   t1[3799] := 0.1576416;
   t1[3800] := 0.1064425;
   t1[3801] := 0.0526067;
   t1[3802] := -0.0066586;
   t1[3803] := -0.0740744;
   t1[3804] := -0.1487714;
   t1[3805] := -0.2246916;
   t1[3806] := -0.2953722;
   t1[3807] := -0.3543501;
   t1[3808] := -0.3951623;
   t1[3809] := -0.4124203;
   t1[3810] := 0.2382786;
   t1[3811] := 0.2234323;
   t1[3812] := 0.2057212;
   t1[3813] := 0.1861852;
   t1[3814] := 0.1646943;
   t1[3815] := 0.1407051;
   t1[3816] := 0.1136735;
   t1[3817] := 0.0830556;
   t1[3818] := 0.0483291;
   t1[3819] := 0.0100414;
   t1[3820] := -0.0297129;
   t1[3821] := -0.0687187;
   t1[3822] := -0.1047607;
   t1[3823] := -0.1356239;
   t1[3824] := -0.1593218;
   t1[3825] := 0.0314255;
   t1[3826] := 0.0159087;
   t1[3827] := 0.0083954;
   t1[3828] := 0.0117159;
   t1[3829] := 0.0246836;
   t1[3830] := 0.0446926;
   t1[3831] := 0.0691354;
   t1[3832] := 0.0954045;
   t1[3833] := 0.1209108;
   t1[3834] := 0.1439967;
   t1[3835] := 0.1643503;
   t1[3836] := 0.1817647;
   t1[3837] := 0.1960331;
   t1[3838] := 0.2069486;
   t1[3839] := 0.2142785;
   t1[3840] := 0.0667891;
   t1[3841] := 0.0459893;
   t1[3842] := 0.0290749;
   t1[3843] := 0.0181673;
   t1[3844] := 0.0125522;
   t1[3845] := 0.0105136;
   t1[3846] := 0.010334;
   t1[3847] := 0.0102961;
   t1[3848] := 0.0087127;
   t1[3849] := 0.0054041;
   t1[3850] := 0.0023689;
   t1[3851] := 0.0017762;
   t1[3852] := 0.0057949;
   t1[3853] := 0.0165937;
   t1[3854] := 0.0358182;
   t1[3855] := -0.1236024;
   t1[3856] := -0.1436511;
   t1[3857] := -0.1554508;
   t1[3858] := -0.1564814;
   t1[3859] := -0.1472676;
   t1[3860] := -0.1294098;
   t1[3861] := -0.1045099;
   t1[3862] := -0.0741695;
   t1[3863] := -0.0400035;
   t1[3864] := -0.0042752;
   t1[3865] := 0.029814;
   t1[3866] := 0.05899;
   t1[3867] := 0.0799781;
   t1[3868] := 0.0895042;
   t1[3869] := 0.0849915;
   t1[3870] := 0.1448045;
   t1[3871] := 0.1536896;
   t1[3872] := 0.1602021;
   t1[3873] := 0.1635016;
   t1[3874] := 0.1634868;
   t1[3875] := 0.1603173;
   t1[3876] := 0.1541528;
   t1[3877] := 0.1451532;
   t1[3878] := 0.1334766;
   t1[3879] := 0.1191958;
   t1[3880] := 0.1022594;
   t1[3881] := 0.0826069;
   t1[3882] := 0.0601774;
   t1[3883] := 0.0349101;
   t1[3884] := 0.0069634;
   t1[3885] := 0.0060057;
   t1[3886] := -0.002674;
   t1[3887] := -0.0069002;
   t1[3888] := -0.0053898;
   t1[3889] := 0.001487;
   t1[3890] := 0.0127761;
   t1[3891] := 0.0275223;
   t1[3892] := 0.0447709;
   t1[3893] := 0.063564;
   t1[3894] := 0.0828049;
   t1[3895] := 0.1011957;
   t1[3896] := 0.1174229;
   t1[3897] := 0.130173;
   t1[3898] := 0.1381326;
   t1[3899] := 0.1401622;
   t1[3900] := 0.1874084;
   t1[3901] := 0.1562083;
   t1[3902] := 0.1240833;
   t1[3903] := 0.0933504;
   t1[3904] := 0.0642;
   t1[3905] := 0.0360715;
   t1[3906] := 0.0084033;
   t1[3907] := -0.0193662;
   t1[3908] := -0.0477891;
   t1[3909] := -0.0769431;
   t1[3910] := -0.1062206;
   t1[3911] := -0.1349603;
   t1[3912] := -0.162501;
   t1[3913] := -0.1881814;
   t1[3914] := -0.2112326;
   t1[3915] := -0.0535974;
   t1[3916] := -0.0502168;
   t1[3917] := -0.0400993;
   t1[3918] := -0.0239367;
   t1[3919] := -0.0041446;
   t1[3920] := 0.0162519;
   t1[3921] := 0.0342271;
   t1[3922] := 0.0467551;
   t1[3923] := 0.0508583;
   t1[3924] := 0.0459583;
   t1[3925] := 0.0349444;
   t1[3926] := 0.0209767;
   t1[3927] := 0.0072152;
   t1[3928] := -0.0031799;
   t1[3929] := -0.0075761;
   t1[3930] := 0.1498998;
   t1[3931] := 0.130271;
   t1[3932] := 0.107127;
   t1[3933] := 0.0806729;
   t1[3934] := 0.052375;
   t1[3935] := 0.0241449;
   t1[3936] := -0.0021051;
   t1[3937] := -0.0244629;
   t1[3938] := -0.0410386;
   t1[3939] := -0.0510728;
   t1[3940] := -0.0554392;
   t1[3941] := -0.055139;
   t1[3942] := -0.0511733;
   t1[3943] := -0.0445433;
   t1[3944] := -0.0362266;
   t1[3945] := -0.2330382;
   t1[3946] := -0.1871568;
   t1[3947] := -0.1450667;
   t1[3948] := -0.1113965;
   t1[3949] := -0.0854538;
   t1[3950] := -0.0646658;
   t1[3951] := -0.0464576;
   t1[3952] := -0.0282541;
   t1[3953] := -0.0075134;
   t1[3954] := 0.0166584;
   t1[3955] := 0.0427734;
   t1[3956] := 0.0691579;
   t1[3957] := 0.0941378;
   t1[3958] := 0.1160396;
   t1[3959] := 0.1332923;
   t1[3960] := -0.0491654;
   t1[3961] := -0.036231;
   t1[3962] := -0.0223325;
   t1[3963] := -0.0065351;
   t1[3964] := 0.0112607;
   t1[3965] := 0.0308597;
   t1[3966] := 0.0520663;
   t1[3967] := 0.0746847;
   t1[3968] := 0.0985081;
   t1[3969] := 0.1227671;
   t1[3970] := 0.1458796;
   t1[3971] := 0.1662;
   t1[3972] := 0.1820826;
   t1[3973] := 0.1918821;
   t1[3974] := 0.1942146;
   t1[3975] := -0.0419469;
   t1[3976] := -0.024382;
   t1[3977] := -0.0039275;
   t1[3978] := 0.0193405;
   t1[3979] := 0.043617;
   t1[3980] := 0.0664858;
   t1[3981] := 0.0855298;
   t1[3982] := 0.0983321;
   t1[3983] := 0.1025108;
   t1[3984] := 0.0974387;
   t1[3985] := 0.0850243;
   t1[3986] := 0.0673741;
   t1[3987] := 0.0465946;
   t1[3988] := 0.0247923;
   t1[3989] := 0.0039388;
   t1[3990] := 0.081306;
   t1[3991] := 0.0967213;
   t1[3992] := 0.1059721;
   t1[3993] := 0.105438;
   t1[3994] := 0.0966705;
   t1[3995] := 0.0830483;
   t1[3996] := 0.067952;
   t1[3997] := 0.0547624;
   t1[3998] := 0.0468165;
   t1[3999] := 0.0452519;
   t1[4000] := 0.0480284;
   t1[4001] := 0.0528576;
   t1[4002] := 0.0574511;
   t1[4003] := 0.0595205;
   t1[4004] := 0.0571091;
   t1[4005] := -0.3532258;
   t1[4006] := -0.347388;
   t1[4007] := -0.3259861;
   t1[4008] := -0.2866082;
   t1[4009] := -0.2320336;
   t1[4010] := -0.1668758;
   t1[4011] := -0.0957504;
   t1[4012] := -0.023273;
   t1[4013] := 0.0459573;
   t1[4014] := 0.1081692;
   t1[4015] := 0.1607873;
   t1[4016] := 0.2013298;
   t1[4017] := 0.2273147;
   t1[4018] := 0.2362603;
   t1[4019] := 0.2265386;
   t1[4020] := -0.1837068;
   t1[4021] := -0.1607816;
   t1[4022] := -0.1328929;
   t1[4023] := -0.1009052;
   t1[4024] := -0.066294;
   t1[4025] := -0.0307508;
   t1[4026] := 0.004033;
   t1[4027] := 0.0363657;
   t1[4028] := 0.064572;
   t1[4029] := 0.0877905;
   t1[4030] := 0.1063364;
   t1[4031] := 0.1206166;
   t1[4032] := 0.1310381;
   t1[4033] := 0.1380079;
   t1[4034] := 0.1419902;
   t1[4035] := 0.1791124;
   t1[4036] := 0.1800564;
   t1[4037] := 0.179791;
   t1[4038] := 0.1790846;
   t1[4039] := 0.1772211;
   t1[4040] := 0.1729594;
   t1[4041] := 0.1650582;
   t1[4042] := 0.1522758;
   t1[4043] := 0.133402;
   t1[4044] := 0.1087973;
   t1[4045] := 0.0810914;
   t1[4046] := 0.0530913;
   t1[4047] := 0.027604;
   t1[4048] := 0.0074365;
   t1[4049] := -0.0050674;
   t1[4050] := 0.18974;
   t1[4051] := 0.1681934;
   t1[4052] := 0.1429099;
   t1[4053] := 0.115058;
   t1[4054] := 0.0845972;
   t1[4055] := 0.0510596;
   t1[4056] := 0.0139768;
   t1[4057] := -0.0271196;
   t1[4058] := -0.0726646;
   t1[4059] := -0.1214214;
   t1[4060] := -0.1697376;
   t1[4061] := -0.2137718;
   t1[4062] := -0.249683;
   t1[4063] := -0.27363;
   t1[4064] := -0.282454;
   t1[4065] := -0.0203979;
   t1[4066] := -0.0223091;
   t1[4067] := -0.0231968;
   t1[4068] := -0.0224718;
   t1[4069] := -0.0193559;
   t1[4070] := -0.0130042;
   t1[4071] := -0.0025716;
   t1[4072] := 0.012787;
   t1[4073] := 0.0338832;
   t1[4074] := 0.05985;
   t1[4075] := 0.0873946;
   t1[4076] := 0.113035;
   t1[4077] := 0.1332889;
   t1[4078] := 0.1446745;
   t1[4079] := 0.1443445;
   t1[4080] := 0.058554;
   t1[4081] := 0.0751369;
   t1[4082] := 0.0861599;
   t1[4083] := 0.0897582;
   t1[4084] := 0.0872719;
   t1[4085] := 0.0811738;
   t1[4086] := 0.0739379;
   t1[4087] := 0.0680383;
   t1[4088] := 0.0659192;
   t1[4089] := 0.068534;
   t1[4090] := 0.0746809;
   t1[4091] := 0.0829904;
   t1[4092] := 0.0920926;
   t1[4093] := 0.1006178;
   t1[4094] := 0.1072876;
   t1[4095] := -0.1914829;
   t1[4096] := -0.137766;
   t1[4097] := -0.0834525;
   t1[4098] := -0.0324906;
   t1[4099] := 0.0136321;
   t1[4100] := 0.0542972;
   t1[4101] := 0.0888875;
   t1[4102] := 0.1167857;
   t1[4103] := 0.1373913;
   t1[4104] := 0.1509367;
   t1[4105] := 0.1588583;
   t1[4106] := 0.1626864;
   t1[4107] := 0.1639515;
   t1[4108] := 0.164184;
   t1[4109] := 0.1646439;
   t1[4110] := -0.0583478;
   t1[4111] := -0.0186663;
   t1[4112] := 0.0169952;
   t1[4113] := 0.04533;
   t1[4114] := 0.0669303;
   t1[4115] := 0.0837658;
   t1[4116] := 0.0978078;
   t1[4117] := 0.1110275;
   t1[4118] := 0.1253682;
   t1[4119] := 0.1413658;
   t1[4120] := 0.1575224;
   t1[4121] := 0.1721816;
   t1[4122] := 0.1836867;
   t1[4123] := 0.1903812;
   t1[4124] := 0.190859;
   t1[4125] := -0.0328098;
   t1[4126] := -0.0068127;
   t1[4127] := 0.0114748;
   t1[4128] := 0.0191703;
   t1[4129] := 0.0181671;
   t1[4130] := 0.0120459;
   t1[4131] := 0.0043894;
   t1[4132] := -0.0012196;
   t1[4133] := -0.0012441;
   t1[4134] := 0.0055699;
   t1[4135] := 0.0171766;
   t1[4136] := 0.0312727;
   t1[4137] := 0.0455549;
   t1[4138] := 0.05772;
   t1[4139] := 0.0657464;
   t1[4140] := 0.0864437;
   t1[4141] := 0.0887006;
   t1[4142] := 0.0839517;
   t1[4143] := 0.0726865;
   t1[4144] := 0.0565655;
   t1[4145] := 0.0376631;
   t1[4146] := 0.018054;
   t1[4147] := -0.0001868;
   t1[4148] := -0.0150103;
   t1[4149] := -0.0256528;
   t1[4150] := -0.0332085;
   t1[4151] := -0.0389166;
   t1[4152] := -0.0440164;
   t1[4153] := -0.049747;
   t1[4154] := -0.0571015;
   t1[4155] := -0.0806194;
   t1[4156] := -0.0510695;
   t1[4157] := -0.0227195;
   t1[4158] := 0.0029388;
   t1[4159] := 0.0255656;
   t1[4160] := 0.0452287;
   t1[4161] := 0.0619963;
   t1[4162] := 0.0759363;
   t1[4163] := 0.0871133;
   t1[4164] := 0.0954085;
   t1[4165] := 0.1004382;
   t1[4166] := 0.1017982;
   t1[4167] := 0.0990841;
   t1[4168] := 0.0918918;
   t1[4169] := 0.080022;
   t1[4170] := 0.0758055;
   t1[4171] := 0.0483579;
   t1[4172] := 0.019726;
   t1[4173] := -0.0085936;
   t1[4174] := -0.0351953;
   t1[4175] := -0.0587056;
   t1[4176] := -0.0777511;
   t1[4177] := -0.0909582;
   t1[4178] := -0.0969803;
   t1[4179] := -0.0958076;
   t1[4180] := -0.0893632;
   t1[4181] := -0.0797205;
   t1[4182] := -0.0689533;
   t1[4183] := -0.0591352;
   t1[4184] := -0.0520488;
   t1[4185] := 0.0500193;
   t1[4186] := 0.0250257;
   t1[4187] := 0.0067496;
   t1[4188] := -0.0013496;
   t1[4189] := -0.0002283;
   t1[4190] := 0.0075968;
   t1[4191] := 0.0196071;
   t1[4192] := 0.0332839;
   t1[4193] := 0.0461257;
   t1[4194] := 0.0564741;
   t1[4195] := 0.06389;
   t1[4196] := 0.0680293;
   t1[4197] := 0.0685479;
   t1[4198] := 0.0651018;
   t1[4199] := 0.0575236;
   t1[4200] := -0.1111487;
   t1[4201] := -0.1043046;
   t1[4202] := -0.0834341;
   t1[4203] := -0.0456349;
   t1[4204] := 0.0052346;
   t1[4205] := 0.0629264;
   t1[4206] := 0.1211901;
   t1[4207] := 0.1737752;
   t1[4208] := 0.2144941;
   t1[4209] := 0.2403017;
   t1[4210] := 0.2526951;
   t1[4211] := 0.2535257;
   t1[4212] := 0.2446451;
   t1[4213] := 0.2279048;
   t1[4214] := 0.2051906;
   t1[4215] := -0.1796006;
   t1[4216] := -0.1449579;
   t1[4217] := -0.1035627;
   t1[4218] := -0.0561289;
   t1[4219] := -0.0046341;
   t1[4220] := 0.0484977;
   t1[4221] := 0.1008417;
   t1[4222] := 0.1499734;
   t1[4223] := 0.1934813;
   t1[4224] := 0.229624;
   t1[4225] := 0.2576274;
   t1[4226] := 0.2767932;
   t1[4227] := 0.2864232;
   t1[4228] := 0.285819;
   t1[4229] := 0.2745421;
   t1[4230] := -0.1943461;
   t1[4231] := -0.1704851;
   t1[4232] := -0.1405829;
   t1[4233] := -0.1052732;
   t1[4234] := -0.0649546;
   t1[4235] := -0.0199427;
   t1[4236] := 0.0294473;
   t1[4237] := 0.0828997;
   t1[4238] := 0.1400708;
   t1[4239] := 0.1992041;
   t1[4240] := 0.2565007;
   t1[4241] := 0.3080023;
   t1[4242] := 0.3497505;
   t1[4243] := 0.3777874;
   t1[4244] := 0.3887276;
   t1[4245] := 0.1895632;
   t1[4246] := 0.1862952;
   t1[4247] := 0.1769894;
   t1[4248] := 0.1617853;
   t1[4249] := 0.1431127;
   t1[4250] := 0.1242102;
   t1[4251] := 0.1083174;
   t1[4252] := 0.0986739;
   t1[4253] := 0.0984564;
   t1[4254] := 0.1076931;
   t1[4255] := 0.1218616;
   t1[4256] := 0.1360845;
   t1[4257] := 0.145484;
   t1[4258] := 0.1451829;
   t1[4259] := 0.1312412;
   t1[4260] := -0.0941189;
   t1[4261] := -0.0750441;
   t1[4262] := -0.0494044;
   t1[4263] := -0.0175561;
   t1[4264] := 0.018117;
   t1[4265] := 0.0545142;
   t1[4266] := 0.0885344;
   t1[4267] := 0.117076;
   t1[4268] := 0.1370689;
   t1[4269] := 0.1470022;
   t1[4270] := 0.1476181;
   t1[4271] := 0.1398349;
   t1[4272] := 0.1245708;
   t1[4273] := 0.1027442;
   t1[4274] := 0.0753431;
   t1[4275] := 0.0685778;
   t1[4276] := 0.051928;
   t1[4277] := 0.0314925;
   t1[4278] := 0.007498;
   t1[4279] := -0.0187296;
   t1[4280] := -0.0454757;
   t1[4281] := -0.0710255;
   t1[4282] := -0.0936643;
   t1[4283] := -0.1116789;
   t1[4284] := -0.1234511;
   t1[4285] := -0.1274992;
   t1[4286] := -0.1223522;
   t1[4287] := -0.106539;
   t1[4288] := -0.0785887;
   t1[4289] := -0.0377033;
   t1[4290] := -0.1350671;
   t1[4291] := -0.1060196;
   t1[4292] := -0.0778034;
   t1[4293] := -0.0545455;
   t1[4294] := -0.0360641;
   t1[4295] := -0.020655;
   t1[4296] := -0.0066124;
   t1[4297] := 0.0077697;
   t1[4298] := 0.0241794;
   t1[4299] := 0.043411;
   t1[4300] := 0.0649677;
   t1[4301] := 0.0882515;
   t1[4302] := 0.1126646;
   t1[4303] := 0.1376094;
   t1[4304] := 0.1623792;
   t1[4305] := -0.0144924;
   t1[4306] := -0.0096911;
   t1[4307] := -0.00347;
   t1[4308] := 0.0033079;
   t1[4309] := 0.0099354;
   t1[4310] := 0.0157605;
   t1[4311] := 0.0201311;
   t1[4312] := 0.022395;
   t1[4313] := 0.0219254;
   t1[4314] := 0.0193535;
   t1[4315] := 0.0171285;
   t1[4316] := 0.0178418;
   t1[4317] := 0.0240846;
   t1[4318] := 0.0384482;
   t1[4319] := 0.0627826;
   t1[4320] := -0.1042536;
   t1[4321] := -0.0667104;
   t1[4322] := -0.0323665;
   t1[4323] := -0.0045362;
   t1[4324] := 0.017397;
   t1[4325] := 0.0354384;
   t1[4326] := 0.0515946;
   t1[4327] := 0.0678727;
   t1[4328] := 0.0862458;
   t1[4329] := 0.1070016;
   t1[4330] := 0.1279919;
   t1[4331] := 0.1468786;
   t1[4332] := 0.1613233;
   t1[4333] := 0.1689879;
   t1[4334] := 0.1679946;
   t1[4335] := 0.0434848;
   t1[4336] := 0.0531504;
   t1[4337] := 0.0601945;
   t1[4338] := 0.0632927;
   t1[4339] := 0.0616237;
   t1[4340] := 0.0545442;
   t1[4341] := 0.0414107;
   t1[4342] := 0.0215801;
   t1[4343] := -0.0055602;
   t1[4344] := -0.0390802;
   t1[4345] := -0.0758206;
   t1[4346] := -0.1124483;
   t1[4347] := -0.1456301;
   t1[4348] := -0.1720328;
   t1[4349] := -0.1887759;
   t1[4350] := -0.0447853;
   t1[4351] := -0.0387455;
   t1[4352] := -0.0276729;
   t1[4353] := -0.0104063;
   t1[4354] := 0.0118896;
   t1[4355] := 0.0372285;
   t1[4356] := 0.0636228;
   t1[4357] := 0.0890853;
   t1[4358] := 0.1116374;
   t1[4359] := 0.1297481;
   t1[4360] := 0.1425325;
   t1[4361] := 0.1491565;
   t1[4362] := 0.1487859;
   t1[4363] := 0.1405863;
   t1[4364] := 0.1241035;
   t1[4365] := 0.1752176;
   t1[4366] := 0.1764574;
   t1[4367] := 0.1733454;
   t1[4368] := 0.166352;
   t1[4369] := 0.1567683;
   t1[4370] := 0.1461753;
   t1[4371] := 0.1361545;
   t1[4372] := 0.1282874;
   t1[4373] := 0.1241305;
   t1[4374] := 0.1239933;
   t1[4375] := 0.1263832;
   t1[4376] := 0.1296669;
   t1[4377] := 0.1322112;
   t1[4378] := 0.1323828;
   t1[4379] := 0.1288362;
   t1[4380] := 0.1311117;
   t1[4381] := 0.1251942;
   t1[4382] := 0.1175675;
   t1[4383] := 0.1089724;
   t1[4384] := 0.100168;
   t1[4385] := 0.0919197;
   t1[4386] := 0.084993;
   t1[4387] := 0.0801534;
   t1[4388] := 0.0781383;
   t1[4389] := 0.0782922;
   t1[4390] := 0.0779461;
   t1[4391] := 0.0742737;
   t1[4392] := 0.0644488;
   t1[4393] := 0.0456451;
   t1[4394] := 0.015853;
   t1[4395] := 0.1653865;
   t1[4396] := 0.1615747;
   t1[4397] := 0.1489204;
   t1[4398] := 0.1252114;
   t1[4399] := 0.0928236;
   t1[4400] := 0.0557549;
   t1[4401] := 0.0180047;
   t1[4402] := -0.0164276;
   t1[4403] := -0.0435795;
   t1[4404] := -0.061344;
   t1[4405] := -0.0702954;
   t1[4406] := -0.0712172;
   t1[4407] := -0.0648929;
   t1[4408] := -0.0521063;
   t1[4409] := -0.033843;
   t1[4410] := -0.1095109;
   t1[4411] := -0.1050676;
   t1[4412] := -0.0937962;
   t1[4413] := -0.0753762;
   t1[4414] := -0.0512059;
   t1[4415] := -0.0232909;
   t1[4416] := 0.0063625;
   t1[4417] := 0.0357481;
   t1[4418] := 0.0628728;
   t1[4419] := 0.0864108;
   t1[4420] := 0.1059999;
   t1[4421] := 0.1213535;
   t1[4422] := 0.1321848;
   t1[4423] := 0.1382072;
   t1[4424] := 0.1392217;
   t1[4425] := 0.1267594;
   t1[4426] := 0.1530687;
   t1[4427] := 0.1682366;
   t1[4428] := 0.1672206;
   t1[4429] := 0.1514878;
   t1[4430] := 0.1248052;
   t1[4431] := 0.0909425;
   t1[4432] := 0.0536695;
   t1[4433] := 0.0167313;
   t1[4434] := -0.0173527;
   t1[4435] := -0.047835;
   t1[4436] := -0.0741062;
   t1[4437] := -0.0955572;
   t1[4438] := -0.1115787;
   t1[4439] := -0.121677;
   t1[4440] := 0.0897872;
   t1[4441] := 0.0856847;
   t1[4442] := 0.0806051;
   t1[4443] := 0.0744163;
   t1[4444] := 0.0680452;
   t1[4445] := 0.0627932;
   t1[4446] := 0.0599619;
   t1[4447] := 0.060853;
   t1[4448] := 0.0667383;
   t1[4449] := 0.0773905;
   t1[4450] := 0.0904158;
   t1[4451] := 0.1032513;
   t1[4452] := 0.113334;
   t1[4453] := 0.1181012;
   t1[4454] := 0.115397;
   t1[4455] := 0.1432041;
   t1[4456] := 0.1568891;
   t1[4457] := 0.1634402;
   t1[4458] := 0.1613314;
   t1[4459] := 0.1513807;
   t1[4460] := 0.1352343;
   t1[4461] := 0.1145394;
   t1[4462] := 0.0909433;
   t1[4463] := 0.0660909;
   t1[4464] := 0.0415152;
   t1[4465] := 0.0185874;
   t1[4466] := -0.0013338;
   t1[4467] := -0.0168899;
   t1[4468] := -0.0267222;
   t1[4469] := -0.0297787;
   t1[4470] := -0.3758105;
   t1[4471] := -0.322452;
   t1[4472] := -0.2597182;
   t1[4473] := -0.1912154;
   t1[4474] := -0.1200375;
   t1[4475] := -0.049098;
   t1[4476] := 0.0186902;
   t1[4477] := 0.080414;
   t1[4478] := 0.1331862;
   t1[4479] := 0.1754149;
   t1[4480] := 0.20738;
   t1[4481] := 0.2295079;
   t1[4482] := 0.2422246;
   t1[4483] := 0.2459562;
   t1[4484] := 0.2412414;
   t1[4485] := -0.083162;
   t1[4486] := -0.068404;
   t1[4487] := -0.051038;
   t1[4488] := -0.032456;
   t1[4489] := -0.0130457;
   t1[4490] := 0.00716;
   t1[4491] := 0.0281286;
   t1[4492] := 0.0498277;
   t1[4493] := 0.072215;
   t1[4494] := 0.094764;
   t1[4495] := 0.1162474;
   t1[4496] := 0.1353838;
   t1[4497] := 0.1508913;
   t1[4498] := 0.1614884;
   t1[4499] := 0.1660409;
   t1[4500] := 0.1987849;
   t1[4501] := 0.1696371;
   t1[4502] := 0.1381494;
   t1[4503] := 0.1057929;
   t1[4504] := 0.0741976;
   t1[4505] := 0.0450496;
   t1[4506] := 0.0200352;
   t1[4507] := 0.0008408;
   t1[4508] := -0.010889;
   t1[4509] := -0.0155813;
   t1[4510] := -0.0166583;
   t1[4511] := -0.017776;
   t1[4512] := -0.0225902;
   t1[4513] := -0.0347571;
   t1[4514] := -0.0570455;
   t1[4515] := 0.0881659;
   t1[4516] := 0.0702802;
   t1[4517] := 0.0476581;
   t1[4518] := 0.0215006;
   t1[4519] := -0.0062864;
   t1[4520] := -0.0335475;
   t1[4521] := -0.0581276;
   t1[4522] := -0.077871;
   t1[4523] := -0.0906534;
   t1[4524] := -0.0959001;
   t1[4525] := -0.0952757;
   t1[4526] := -0.0906199;
   t1[4527] := -0.0837726;
   t1[4528] := -0.0765732;
   t1[4529] := -0.0706219;
   t1[4530] := 0.2818092;
   t1[4531] := 0.2552775;
   t1[4532] := 0.210369;
   t1[4533] := 0.144979;
   t1[4534] := 0.0648285;
   t1[4535] := -0.0215958;
   t1[4536] := -0.1058042;
   t1[4537] := -0.179307;
   t1[4538] := -0.2337158;
   t1[4539] := -0.265707;
   t1[4540] := -0.2792773;
   t1[4541] := -0.2789946;
   t1[4542] := -0.2694269;
   t1[4543] := -0.2551424;
   t1[4544] := -0.2401939;
   t1[4545] := 0.2836724;
   t1[4546] := 0.24923;
   t1[4547] := 0.2094985;
   t1[4548] := 0.1652706;
   t1[4549] := 0.1183369;
   t1[4550] := 0.0708402;
   t1[4551] := 0.0249238;
   t1[4552] := -0.017269;
   t1[4553] := -0.0536144;
   t1[4554] := -0.0829686;
   t1[4555] := -0.1056038;
   t1[4556] := -0.1219029;
   t1[4557] := -0.1322485;
   t1[4558] := -0.1370237;
   t1[4559] := -0.1366486;
   t1[4560] := 0.0013929;
   t1[4561] := -0.0233614;
   t1[4562] := -0.0422055;
   t1[4563] := -0.0543371;
   t1[4564] := -0.0599601;
   t1[4565] := -0.0596343;
   t1[4566] := -0.0539198;
   t1[4567] := -0.0433767;
   t1[4568] := -0.0285641;
   t1[4569] := -0.0099806;
   t1[4570] := 0.0119624;
   t1[4571] := 0.0368602;
   t1[4572] := 0.0643079;
   t1[4573] := 0.093901;
   t1[4574] := 0.1249875;
   t1[4575] := 0.2746963;
   t1[4576] := 0.2280546;
   t1[4577] := 0.1791329;
   t1[4578] := 0.1300266;
   t1[4579] := 0.0810237;
   t1[4580] := 0.0317734;
   t1[4581] := -0.0180759;
   t1[4582] := -0.0688756;
   t1[4583] := -0.1209428;
   t1[4584] := -0.1728681;
   t1[4585] := -0.220747;
   t1[4586] := -0.2604801;
   t1[4587] := -0.2879682;
   t1[4588] := -0.299112;
   t1[4589] := -0.2907236;
   t1[4590] := 0.227914;
   t1[4591] := 0.2009724;
   t1[4592] := 0.1743917;
   t1[4593] := 0.1505338;
   t1[4594] := 0.130849;
   t1[4595] := 0.1164656;
   t1[4596] := 0.1085113;
   t1[4597] := 0.108114;
   t1[4598] := 0.1163595;
   t1[4599] := 0.1322398;
   t1[4600] := 0.1517199;
   t1[4601] := 0.1705288;
   t1[4602] := 0.1843953;
   t1[4603] := 0.1890485;
   t1[4604] := 0.1810103;
   t1[4605] := -0.0870302;
   t1[4606] := -0.0465301;
   t1[4607] := -0.0089114;
   t1[4608] := 0.0220016;
   t1[4609] := 0.0460928;
   t1[4610] := 0.0645562;
   t1[4611] := 0.0785875;
   t1[4612] := 0.0893821;
   t1[4613] := 0.0981219;
   t1[4614] := 0.1052981;
   t1[4615] := 0.1104034;
   t1[4616] := 0.1128528;
   t1[4617] := 0.1120614;
   t1[4618] := 0.1074442;
   t1[4619] := 0.0986109;
   t1[4620] := -0.1728606;
   t1[4621] := -0.127203;
   t1[4622] := -0.0755065;
   t1[4623] := -0.020009;
   t1[4624] := 0.0368642;
   t1[4625] := 0.0926215;
   t1[4626] := 0.1447711;
   t1[4627] := 0.1908214;
   t1[4628] := 0.2283021;
   t1[4629] := 0.2558181;
   t1[4630] := 0.2735277;
   t1[4631] := 0.2817105;
   t1[4632] := 0.2806462;
   t1[4633] := 0.2706145;
   t1[4634] := 0.2520499;
   t1[4635] := -0.1085393;
   t1[4636] := -0.0655247;
   t1[4637] := -0.0193889;
   t1[4638] := 0.0274051;
   t1[4639] := 0.0730157;
   t1[4640] := 0.1158207;
   t1[4641] := 0.1541983;
   t1[4642] := 0.1865267;
   t1[4643] := 0.2112014;
   t1[4644] := 0.2274901;
   t1[4645] := 0.2359207;
   t1[4646] := 0.2371196;
   t1[4647] := 0.231713;
   t1[4648] := 0.2203275;
   t1[4649] := 0.2035683;
   t1[4650] := 0.0107215;
   t1[4651] := 0.0308927;
   t1[4652] := 0.0446619;
   t1[4653] := 0.0494573;
   t1[4654] := 0.0477508;
   t1[4655] := 0.0437966;
   t1[4656] := 0.0418509;
   t1[4657] := 0.0461699;
   t1[4658] := 0.0609356;
   t1[4659] := 0.0866115;
   t1[4660] := 0.1182874;
   t1[4661] := 0.1506335;
   t1[4662] := 0.1783202;
   t1[4663] := 0.1960177;
   t1[4664] := 0.1991685;
   t1[4665] := 0.1538821;
   t1[4666] := 0.1553968;
   t1[4667] := 0.1589691;
   t1[4668] := 0.1654171;
   t1[4669] := 0.1737123;
   t1[4670] := 0.1821734;
   t1[4671] := 0.1891185;
   t1[4672] := 0.1928656;
   t1[4673] := 0.1917473;
   t1[4674] := 0.1848124;
   t1[4675] := 0.1721455;
   t1[4676] := 0.1539121;
   t1[4677] := 0.1302776;
   t1[4678] := 0.1014076;
   t1[4679] := 0.0677879;
   t1[4680] := 0.0969475;
   t1[4681] := 0.0971912;
   t1[4682] := 0.0972052;
   t1[4683] := 0.0969806;
   t1[4684] := 0.0971251;
   t1[4685] := 0.0984642;
   t1[4686] := 0.1018237;
   t1[4687] := 0.1080296;
   t1[4688] := 0.1178736;
   t1[4689] := 0.1304501;
   t1[4690] := 0.1424002;
   t1[4691] := 0.1501734;
   t1[4692] := 0.1502191;
   t1[4693] := 0.138987;
   t1[4694] := 0.113698;
   t1[4695] := 0.1916815;
   t1[4696] := 0.1797811;
   t1[4697] := 0.1629954;
   t1[4698] := 0.1418429;
   t1[4699] := 0.1177478;
   t1[4700] := 0.0924546;
   t1[4701] := 0.0677081;
   t1[4702] := 0.045253;
   t1[4703] := 0.0268173;
   t1[4704] := 0.0132891;
   t1[4705] := 0.0043422;
   t1[4706] := -0.0004442;
   t1[4707] := -0.0014908;
   t1[4708] := 0.0007814;
   t1[4709] := 0.0059547;
   t1[4710] := 0.0511631;
   t1[4711] := 0.0523964;
   t1[4712] := 0.0471871;
   t1[4713] := 0.0346185;
   t1[4714] := 0.0172187;
   t1[4715] := -0.001267;
   t1[4716] := -0.017092;
   t1[4717] := -0.0265097;
   t1[4718] := -0.0258269;
   t1[4719] := -0.0140292;
   t1[4720] := 0.0060268;
   t1[4721] := 0.0311822;
   t1[4722] := 0.0582783;
   t1[4723] := 0.0841562;
   t1[4724] := 0.1059692;
   t1[4725] := 0.1451963;
   t1[4726] := 0.1252911;
   t1[4727] := 0.1059383;
   t1[4728] := 0.0896385;
   t1[4729] := 0.0774641;
   t1[4730] := 0.0699829;
   t1[4731] := 0.0677619;
   t1[4732] := 0.0713684;
   t1[4733] := 0.0813547;
   t1[4734] := 0.0975299;
   t1[4735] := 0.1186288;
   t1[4736] := 0.1433028;
   t1[4737] := 0.1702027;
   t1[4738] := 0.1979798;
   t1[4739] := 0.2252449;
   t1[4740] := -0.0490679;
   t1[4741] := -0.0271853;
   t1[4742] := -0.0019549;
   t1[4743] := 0.0256831;
   t1[4744] := 0.0546865;
   t1[4745] := 0.0839769;
   t1[4746] := 0.1124759;
   t1[4747] := 0.139105;
   t1[4748] := 0.162781;
   t1[4749] := 0.1821855;
   t1[4750] := 0.1956595;
   t1[4751] := 0.2015177;
   t1[4752] := 0.1980747;
   t1[4753] := 0.1836451;
   t1[4754] := 0.1571646;
   t1[4755] := 0.1123676;
   t1[4756] := 0.1292125;
   t1[4757] := 0.1436098;
   t1[4758] := 0.1545683;
   t1[4759] := 0.1611561;
   t1[4760] := 0.162462;
   t1[4761] := 0.1575747;
   t1[4762] := 0.1455833;
   t1[4763] := 0.1255971;
   t1[4764] := 0.0977538;
   t1[4765] := 0.0636775;
   t1[4766] := 0.0251082;
   t1[4767] := -0.0162142;
   t1[4768] := -0.0585496;
   t1[4769] := -0.1001368;
   t1[4770] := 0.2482718;
   t1[4771] := 0.2225692;
   t1[4772] := 0.1926065;
   t1[4773] := 0.1580895;
   t1[4774] := 0.1206948;
   t1[4775] := 0.0827955;
   t1[4776] := 0.0467656;
   t1[4777] := 0.014979;
   t1[4778] := -0.0102121;
   t1[4779] := -0.0275512;
   t1[4780] := -0.0373643;
   t1[4781] := -0.0401014;
   t1[4782] := -0.0362123;
   t1[4783] := -0.0261468;
   t1[4784] := -0.010564;
   t1[4785] := 0.2572694;
   t1[4786] := 0.2410908;
   t1[4787] := 0.2268193;
   t1[4788] := 0.2171856;
   t1[4789] := 0.2123168;
   t1[4790] := 0.2114201;
   t1[4791] := 0.2137015;
   t1[4792] := 0.2183671;
   t1[4793] := 0.2246127;
   t1[4794] := 0.2311261;
   t1[4795] := 0.2358603;
   t1[4796] := 0.2367111;
   t1[4797] := 0.2315744;
   t1[4798] := 0.2183459;
   t1[4799] := 0.1955507;
   t1[4800] := 0.0068827;
   t1[4801] := 0.0092901;
   t1[4802] := 0.0146454;
   t1[4803] := 0.0243347;
   t1[4804] := 0.0368081;
   t1[4805] := 0.0494784;
   t1[4806] := 0.0597573;
   t1[4807] := 0.0650564;
   t1[4808] := 0.0628393;
   t1[4809] := 0.0531662;
   t1[4810] := 0.0398507;
   t1[4811] := 0.026999;
   t1[4812] := 0.0187177;
   t1[4813] := 0.0191129;
   t1[4814] := 0.0314385;
   t1[4815] := 0.1902814;
   t1[4816] := 0.1645946;
   t1[4817] := 0.1353592;
   t1[4818] := 0.1037425;
   t1[4819] := 0.071688;
   t1[4820] := 0.0414132;
   t1[4821] := 0.0151362;
   t1[4822] := -0.0049253;
   t1[4823] := -0.0165872;
   t1[4824] := -0.0193721;
   t1[4825] := -0.0152683;
   t1[4826] := -0.0064569;
   t1[4827] := 0.0048812;
   t1[4828] := 0.0165652;
   t1[4829] := 0.0266218;
   t1[4830] := 0.2224702;
   t1[4831] := 0.238518;
   t1[4832] := 0.251734;
   t1[4833] := 0.2614462;
   t1[4834] := 0.2671083;
   t1[4835] := 0.2682182;
   t1[4836] := 0.264274;
   t1[4837] := 0.2547738;
   t1[4838] := 0.2392355;
   t1[4839] := 0.21818;
   t1[4840] := 0.1935769;
   t1[4841] := 0.167509;
   t1[4842] := 0.1420592;
   t1[4843] := 0.1193102;
   t1[4844] := 0.1010374;
   t1[4845] := -0.0465887;
   t1[4846] := -0.0511573;
   t1[4847] := -0.0498118;
   t1[4848] := -0.0414286;
   t1[4849] := -0.0267949;
   t1[4850] := -0.0073737;
   t1[4851] := 0.0153718;
   t1[4852] := 0.0399779;
   t1[4853] := 0.0649816;
   t1[4854] := 0.0889317;
   t1[4855] := 0.110395;
   t1[4856] := 0.1279396;
   t1[4857] := 0.1401335;
   t1[4858] := 0.1455448;
   t1[4859] := 0.14313;
   t1[4860] := 0.0024975;
   t1[4861] := 0.0190176;
   t1[4862] := 0.0423976;
   t1[4863] := 0.0726747;
   t1[4864] := 0.1071544;
   t1[4865] := 0.1421766;
   t1[4866] := 0.1740799;
   t1[4867] := 0.1992031;
   t1[4868] := 0.2139342;
   t1[4869] := 0.217119;
   t1[4870] := 0.2111556;
   t1[4871] := 0.1987192;
   t1[4872] := 0.1824854;
   t1[4873] := 0.1651294;
   t1[4874] := 0.1489674;
   t1[4875] := 0.2869096;
   t1[4876] := 0.2691508;
   t1[4877] := 0.2441442;
   t1[4878] := 0.2113333;
   t1[4879] := 0.1725009;
   t1[4880] := 0.1302561;
   t1[4881] := 0.0872091;
   t1[4882] := 0.0459702;
   t1[4883] := 0.0091329;
   t1[4884] := -0.0215375;
   t1[4885] := -0.0454728;
   t1[4886] := -0.0621983;
   t1[4887] := -0.0712395;
   t1[4888] := -0.0721215;
   t1[4889] := -0.0646722;
   t1[4890] := -0.2695022;
   t1[4891] := -0.2380107;
   t1[4892] := -0.1909814;
   t1[4893] := -0.1288195;
   t1[4894] := -0.0562442;
   t1[4895] := 0.0205009;
   t1[4896] := 0.0951705;
   t1[4897] := 0.1615194;
   t1[4898] := 0.2133677;
   t1[4899] := 0.2478132;
   t1[4900] := 0.2666902;
   t1[4901] := 0.2722028;
   t1[4902] := 0.2665552;
   t1[4903] := 0.2519516;
   t1[4904] := 0.2305451;
   t1[4905] := 0.0727284;
   t1[4906] := 0.0558426;
   t1[4907] := 0.0423075;
   t1[4908] := 0.0344213;
   t1[4909] := 0.0321456;
   t1[4910] := 0.0346163;
   t1[4911] := 0.0409684;
   t1[4912] := 0.0503367;
   t1[4913] := 0.0618536;
   t1[4914] := 0.074514;
   t1[4915] := 0.0871145;
   t1[4916] := 0.0984363;
   t1[4917] := 0.1072607;
   t1[4918] := 0.1123688;
   t1[4919] := 0.1126992;
   t1[4920] := 0.2306891;
   t1[4921] := 0.2132244;
   t1[4922] := 0.1924397;
   t1[4923] := 0.1678365;
   t1[4924] := 0.1399937;
   t1[4925] := 0.1098709;
   t1[4926] := 0.0784282;
   t1[4927] := 0.0466257;
   t1[4928] := 0.0154208;
   t1[4929] := -0.0143669;
   t1[4930] := -0.0421164;
   t1[4931] := -0.0672223;
   t1[4932] := -0.0890794;
   t1[4933] := -0.1070823;
   t1[4934] := -0.1206617;
   t1[4935] := 0.181064;
   t1[4936] := 0.2057841;
   t1[4937] := 0.2246252;
   t1[4938] := 0.2363226;
   t1[4939] := 0.2403454;
   t1[4940] := 0.2364214;
   t1[4941] := 0.224279;
   t1[4942] := 0.2036464;
   t1[4943] := 0.174286;
   t1[4944] := 0.1376635;
   t1[4945] := 0.0977061;
   t1[4946] := 0.0585332;
   t1[4947] := 0.0242643;
   t1[4948] := -0.0009813;
   t1[4949] := -0.0138185;
   t1[4950] := 0.2055318;
   t1[4951] := 0.1693584;
   t1[4952] := 0.1320945;
   t1[4953] := 0.0958028;
   t1[4954] := 0.0619806;
   t1[4955] := 0.0319255;
   t1[4956] := 0.0069349;
   t1[4957] := -0.0116939;
   t1[4958] := -0.0226923;
   t1[4959] := -0.0262294;
   t1[4960] := -0.0245524;
   t1[4961] := -0.0200706;
   t1[4962] := -0.0151934;
   t1[4963] := -0.01233;
   t1[4964] := -0.0134926;
   t1[4965] := 0.2112197;
   t1[4966] := 0.1760574;
   t1[4967] := 0.1421712;
   t1[4968] := 0.1106756;
   t1[4969] := 0.0815539;
   t1[4970] := 0.0543897;
   t1[4971] := 0.0287661;
   t1[4972] := 0.0042661;
   t1[4973] := -0.0195188;
   t1[4974] := -0.0425892;
   t1[4975] := -0.0643556;
   t1[4976] := -0.0841821;
   t1[4977] := -0.1014333;
   t1[4978] := -0.1154734;
   t1[4979] := -0.1257096;
   t1[4980] := -0.0007994;
   t1[4981] := -0.0351105;
   t1[4982] := -0.0597962;
   t1[4983] := -0.0719421;
   t1[4984] := -0.0729129;
   t1[4985] := -0.0655853;
   t1[4986] := -0.0528375;
   t1[4987] := -0.037548;
   t1[4988] := -0.0225699;
   t1[4989] := -0.0094981;
   t1[4990] := 0.0018914;
   t1[4991] := 0.0119643;
   t1[4992] := 0.0210865;
   t1[4993] := 0.0296238;
   t1[4994] := 0.0378596;
   t1[4995] := 0.1402721;
   t1[4996] := 0.1046366;
   t1[4997] := 0.0738667;
   t1[4998] := 0.0498805;
   t1[4999] := 0.0324173;
   t1[5000] := 0.0204463;
   t1[5001] := 0.012936;
   t1[5002] := 0.008855;
   t1[5003] := 0.0071838;
   t1[5004] := 0.0075134;
   t1[5005] := 0.0103166;
   t1[5006] := 0.0161353;
   t1[5007] := 0.0255111;
   t1[5008] := 0.0389858;
   t1[5009] := 0.0567774;
   t1[5010] := 0.2294574;
   t1[5011] := 0.2100077;
   t1[5012] := 0.1906841;
   t1[5013] := 0.172427;
   t1[5014] := 0.1551539;
   t1[5015] := 0.1384207;
   t1[5016] := 0.1217826;
   t1[5017] := 0.1047953;
   t1[5018] := 0.0870206;
   t1[5019] := 0.0683466;
   t1[5020] := 0.0491324;
   t1[5021] := 0.0297743;
   t1[5022] := 0.0106683;
   t1[5023] := -0.0077895;
   t1[5024] := -0.0251548;
   t1[5025] := -0.1089462;
   t1[5026] := -0.056044;
   t1[5027] := -0.0043423;
   t1[5028] := 0.0455206;
   t1[5029] := 0.0931087;
   t1[5030] := 0.1380574;
   t1[5031] := 0.1800023;
   t1[5032] := 0.218579;
   t1[5033] := 0.2534115;
   t1[5034] := 0.2835509;
   t1[5035] := 0.3072199;
   t1[5036] := 0.3225766;
   t1[5037] := 0.3277793;
   t1[5038] := 0.3209861;
   t1[5039] := 0.3009125;
   t1[5040] := 0.3314105;
   t1[5041] := 0.3257191;
   t1[5042] := 0.3094998;
   t1[5043] := 0.2825064;
   t1[5044] := 0.2470406;
   t1[5045] := 0.206305;
   t1[5046] := 0.1635029;
   t1[5047] := 0.1218376;
   t1[5048] := 0.0844692;
   t1[5049] := 0.0523834;
   t1[5050] := 0.0234238;
   t1[5051] := -0.0048114;
   t1[5052] := -0.0347239;
   t1[5053] := -0.0687155;
   t1[5054] := -0.1084454;
   t1[5055] := 0.1738099;
   t1[5056] := 0.1610307;
   t1[5057] := 0.1522964;
   t1[5058] := 0.1498082;
   t1[5059] := 0.151141;
   t1[5060] := 0.152235;
   t1[5061] := 0.1490284;
   t1[5062] := 0.1374595;
   t1[5063] := 0.1135366;
   t1[5064] := 0.0767701;
   t1[5065] := 0.0317313;
   t1[5066] := -0.016613;
   t1[5067] := -0.063296;
   t1[5068] := -0.1033513;
   t1[5069] := -0.1324222;
   t1[5070] := 0.2355668;
   t1[5071] := 0.2226366;
   t1[5072] := 0.2077726;
   t1[5073] := 0.1922539;
   t1[5074] := 0.1759373;
   t1[5075] := 0.1581774;
   t1[5076] := 0.1383279;
   t1[5077] := 0.1157428;
   t1[5078] := 0.0897887;
   t1[5079] := 0.0604747;
   t1[5080] := 0.0287381;
   t1[5081] := -0.0044114;
   t1[5082] := -0.0379638;
   t1[5083] := -0.0709094;
   t1[5084] := -0.1021454;
   t1[5085] := -0.0320041;
   t1[5086] := -0.0399681;
   t1[5087] := -0.0477414;
   t1[5088] := -0.0553136;
   t1[5089] := -0.0606673;
   t1[5090] := -0.0610763;
   t1[5091] := -0.0538133;
   t1[5092] := -0.036151;
   t1[5093] := -0.0054332;
   t1[5094] := 0.0374504;
   t1[5095] := 0.0864851;
   t1[5096] := 0.1352563;
   t1[5097] := 0.177349;
   t1[5098] := 0.2063487;
   t1[5099] := 0.2169217;
   t1[5100] := -0.0383944;
   t1[5101] := -0.0339623;
   t1[5102] := -0.0246457;
   t1[5103] := -0.00961;
   t1[5104] := 0.0099036;
   t1[5105] := 0.0319201;
   t1[5106] := 0.0544638;
   t1[5107] := 0.075559;
   t1[5108] := 0.0932578;
   t1[5109] := 0.1070056;
   t1[5110] := 0.1182613;
   t1[5111] := 0.1286412;
   t1[5112] := 0.1397613;
   t1[5113] := 0.153238;
   t1[5114] := 0.1703339;
   t1[5115] := -0.1165117;
   t1[5116] := -0.0966346;
   t1[5117] := -0.0667644;
   t1[5118] := -0.026801;
   t1[5119] := 0.0198868;
   t1[5120] := 0.0687049;
   t1[5121] := 0.1150574;
   t1[5122] := 0.1543487;
   t1[5123] := 0.1820406;
   t1[5124] := 0.196477;
   t1[5125] := 0.2001663;
   t1[5126] := 0.1959424;
   t1[5127] := 0.1866391;
   t1[5128] := 0.1750901;
   t1[5129] := 0.1636999;
   t1[5130] := 0.0138486;
   t1[5131] := 0.037359;
   t1[5132] := 0.0578786;
   t1[5133] := 0.0725615;
   t1[5134] := 0.0819538;
   t1[5135] := 0.0878004;
   t1[5136] := 0.0918473;
   t1[5137] := 0.0958406;
   t1[5138] := 0.1014977;
   t1[5139] := 0.1090914;
   t1[5140] := 0.1168076;
   t1[5141] := 0.122669;
   t1[5142] := 0.1246985;
   t1[5143] := 0.1209187;
   t1[5144] := 0.1097988;
   t1[5145] := -0.0157056;
   t1[5146] := -0.0322717;
   t1[5147] := -0.0415028;
   t1[5148] := -0.0407201;
   t1[5149] := -0.0310475;
   t1[5150] := -0.0149524;
   t1[5151] := 0.0050964;
   t1[5152] := 0.0266298;
   t1[5153] := 0.0471865;
   t1[5154] := 0.0646902;
   t1[5155] := 0.0776199;
   t1[5156] := 0.0844987;
   t1[5157] := 0.0838491;
   t1[5158] := 0.0741939;
   t1[5159] := 0.0545653;
   t1[5160] := 0.2842315;
   t1[5161] := 0.2918334;
   t1[5162] := 0.2901178;
   t1[5163] := 0.2777814;
   t1[5164] := 0.2556623;
   t1[5165] := 0.225355;
   t1[5166] := 0.1884551;
   t1[5167] := 0.1465583;
   t1[5168] := 0.1012629;
   t1[5169] := 0.0543091;
   t1[5170] := 0.0076422;
   t1[5171] := -0.0367765;
   t1[5172] := -0.0769857;
   t1[5173] := -0.1110242;
   t1[5174] := -0.1371355;
   t1[5175] := 0.0057389;
   t1[5176] := 0.0026206;
   t1[5177] := 0.0018881;
   t1[5178] := 0.0045471;
   t1[5179] := 0.0098998;
   t1[5180] := 0.0166462;
   t1[5181] := 0.023486;
   t1[5182] := 0.0291186;
   t1[5183] := 0.0322621;
   t1[5184] := 0.0325684;
   t1[5185] := 0.0310392;
   t1[5186] := 0.0287812;
   t1[5187] := 0.0269013;
   t1[5188] := 0.0265063;
   t1[5189] := 0.0285084;
   t1[5190] := 0.0366154;
   t1[5191] := 0.0459537;
   t1[5192] := 0.0521963;
   t1[5193] := 0.0530875;
   t1[5194] := 0.0498663;
   t1[5195] := 0.0450063;
   t1[5196] := 0.0409826;
   t1[5197] := 0.0402705;
   t1[5198] := 0.0453039;
   t1[5199] := 0.056456;
   t1[5200] := 0.0711224;
   t1[5201] := 0.0864657;
   t1[5202] := 0.0996488;
   t1[5203] := 0.1078346;
   t1[5204] := 0.1086453;
   t1[5205] := -0.0775259;
   t1[5206] := -0.0428005;
   t1[5207] := -0.006696;
   t1[5208] := 0.029227;
   t1[5209] := 0.063201;
   t1[5210] := 0.0933851;
   t1[5211] := 0.1179383;
   t1[5212] := 0.1350198;
   t1[5213] := 0.1428132;
   t1[5214] := 0.1407407;
   t1[5215] := 0.1300138;
   t1[5216] := 0.111984;
   t1[5217] := 0.0880026;
   t1[5218] := 0.0594208;
   t1[5219] := 0.0276941;
   t1[5220] := -0.1632182;
   t1[5221] := -0.1748871;
   t1[5222] := -0.1808051;
   t1[5223] := -0.1792678;
   t1[5224] := -0.1704627;
   t1[5225] := -0.1552456;
   t1[5226] := -0.134473;
   t1[5227] := -0.1090016;
   t1[5228] := -0.0796864;
   t1[5229] := -0.0473028;
   t1[5230] := -0.0125113;
   t1[5231] := 0.0240365;
   t1[5232] := 0.0616893;
   t1[5233] := 0.0997954;
   t1[5234] := 0.1375059;
   t1[5235] := -0.0010285;
   t1[5236] := 0.0304457;
   t1[5237] := 0.0556515;
   t1[5238] := 0.0716293;
   t1[5239] := 0.0784188;
   t1[5240] := 0.0771191;
   t1[5241] := 0.0688306;
   t1[5242] := 0.0546539;
   t1[5243] := 0.0357047;
   t1[5244] := 0.01387;
   t1[5245] := -0.0078488;
   t1[5246] := -0.0263632;
   t1[5247] := -0.038585;
   t1[5248] := -0.0414257;
   t1[5249] := -0.0325006;
   t1[5250] := 0.1076755;
   t1[5251] := 0.1207554;
   t1[5252] := 0.1317261;
   t1[5253] := 0.1383243;
   t1[5254] := 0.1406147;
   t1[5255] := 0.1394849;
   t1[5256] := 0.1358228;
   t1[5257] := 0.1305169;
   t1[5258] := 0.1244517;
   t1[5259] := 0.1183252;
   t1[5260] := 0.1125663;
   t1[5261] := 0.1075825;
   t1[5262] := 0.1037817;
   t1[5263] := 0.1015714;
   t1[5264] := 0.1011963;
   t1[5265] := -0.1470849;
   t1[5266] := -0.139753;
   t1[5267] := -0.1294944;
   t1[5268] := -0.1153808;
   t1[5269] := -0.0971214;
   t1[5270] := -0.0746503;
   t1[5271] := -0.0479021;
   t1[5272] := -0.0168115;
   t1[5273] := 0.018663;
   t1[5274] := 0.0573512;
   t1[5275] := 0.0963327;
   t1[5276] := 0.1325501;
   t1[5277] := 0.1629464;
   t1[5278] := 0.1844644;
   t1[5279] := 0.1945342;
   t1[5280] := -0.0670065;
   t1[5281] := -0.060024;
   t1[5282] := -0.0527799;
   t1[5283] := -0.0448193;
   t1[5284] := -0.0359242;
   t1[5285] := -0.0259609;
   t1[5286] := -0.0147953;
   t1[5287] := -0.0022938;
   t1[5288] := 0.0116759;
   t1[5289] := 0.0271547;
   t1[5290] := 0.0440527;
   t1[5291] := 0.0622692;
   t1[5292] := 0.081704;
   t1[5293] := 0.1022565;
   t1[5294] := 0.1236341;
   t1[5295] := 0.2054707;
   t1[5296] := 0.1995242;
   t1[5297] := 0.1934798;
   t1[5298] := 0.1879506;
   t1[5299] := 0.1819134;
   t1[5300] := 0.1737664;
   t1[5301] := 0.1619074;
   t1[5302] := 0.1447342;
   t1[5303] := 0.1206806;
   t1[5304] := 0.0899842;
   t1[5305] := 0.0554902;
   t1[5306] := 0.0202471;
   t1[5307] := -0.0126965;
   t1[5308] := -0.0402922;
   t1[5309] := -0.0599163;
   t1[5310] := 0.2266143;
   t1[5311] := 0.1892385;
   t1[5312] := 0.1516248;
   t1[5313] := 0.1177912;
   t1[5314] := 0.0887821;
   t1[5315] := 0.0645915;
   t1[5316] := 0.0452121;
   t1[5317] := 0.0306369;
   t1[5318] := 0.0208476;
   t1[5319] := 0.0152799;
   t1[5320] := 0.0125805;
   t1[5321] := 0.0113342;
   t1[5322] := 0.0101258;
   t1[5323] := 0.0075403;
   t1[5324] := 0.0024472;
   t1[5325] := -0.0377719;
   t1[5326] := -0.0132358;
   t1[5327] := 0.012552;
   t1[5328] := 0.0385148;
   t1[5329] := 0.0641764;
   t1[5330] := 0.0892723;
   t1[5331] := 0.1135382;
   t1[5332] := 0.1367101;
   t1[5333] := 0.1585138;
   t1[5334] := 0.1781882;
   t1[5335] := 0.1942676;
   t1[5336] := 0.2052311;
   t1[5337] := 0.209558;
   t1[5338] := 0.2057278;
   t1[5339] := 0.1925972;
   t1[5340] := 0.0172117;
   t1[5341] := 0.0138449;
   t1[5342] := 0.0055963;
   t1[5343] := -0.0090459;
   t1[5344] := -0.0285871;
   t1[5345] := -0.0504706;
   t1[5346] := -0.0721384;
   t1[5347] := -0.0910323;
   t1[5348] := -0.1046237;
   t1[5349] := -0.1118498;
   t1[5350] := -0.1137662;
   t1[5351] := -0.111594;
   t1[5352] := -0.1065542;
   t1[5353] := -0.0998681;
   t1[5354] := -0.0926496;
   t1[5355] := -0.1580391;
   t1[5356] := -0.0985399;
   t1[5357] := -0.043812;
   t1[5358] := 0.0005705;
   t1[5359] := 0.0349331;
   t1[5360] := 0.0616855;
   t1[5361] := 0.0832402;
   t1[5362] := 0.1020094;
   t1[5363] := 0.1203854;
   t1[5364] := 0.1397596;
   t1[5365] := 0.1600762;
   t1[5366] := 0.1811669;
   t1[5367] := 0.2028631;
   t1[5368] := 0.2249963;
   t1[5369] := 0.2471319;
   t1[5370] := -0.0896867;
   t1[5371] := -0.0488943;
   t1[5372] := -0.0120587;
   t1[5373] := 0.0185452;
   t1[5374] := 0.0429358;
   t1[5375] := 0.061942;
   t1[5376] := 0.0763933;
   t1[5377] := 0.0871195;
   t1[5378] := 0.0949483;
   t1[5379] := 0.1006127;
   t1[5380] := 0.1047086;
   t1[5381] := 0.1078211;
   t1[5382] := 0.1105355;
   t1[5383] := 0.1134371;
   t1[5384] := 0.1169378;
   t1[5385] := 0.0483643;
   t1[5386] := 0.0405087;
   t1[5387] := 0.0357312;
   t1[5388] := 0.0373683;
   t1[5389] := 0.0441397;
   t1[5390] := 0.0531338;
   t1[5391] := 0.0614371;
   t1[5392] := 0.066136;
   t1[5393] := 0.0643667;
   t1[5394] := 0.0557449;
   t1[5395] := 0.0434705;
   t1[5396] := 0.0310232;
   t1[5397] := 0.0218824;
   t1[5398] := 0.0195279;
   t1[5399] := 0.0267103;
   t1[5400] := 0.1923611;
   t1[5401] := 0.1873521;
   t1[5402] := 0.1721971;
   t1[5403] := 0.1463582;
   t1[5404] := 0.1120829;
   t1[5405] := 0.0726028;
   t1[5406] := 0.0311506;
   t1[5407] := -0.009041;
   t1[5408] := -0.0447625;
   t1[5409] := -0.0739701;
   t1[5410] := -0.0963039;
   t1[5411] := -0.1115358;
   t1[5412] := -0.1194375;
   t1[5413] := -0.1197809;
   t1[5414] := -0.1126004;
   t1[5415] := 0.0602888;
   t1[5416] := 0.0781874;
   t1[5417] := 0.0934255;
   t1[5418] := 0.1055462;
   t1[5419] := 0.1142926;
   t1[5420] := 0.1194784;
   t1[5421] := 0.1209173;
   t1[5422] := 0.1184232;
   t1[5423] := 0.1118271;
   t1[5424] := 0.1018268;
   t1[5425] := 0.0903726;
   t1[5426] := 0.0795126;
   t1[5427] := 0.071295;
   t1[5428] := 0.0677678;
   t1[5429] := 0.0704959;
   t1[5430] := 0.0695823;
   t1[5431] := 0.0693244;
   t1[5432] := 0.0733131;
   t1[5433] := 0.0806888;
   t1[5434] := 0.0902777;
   t1[5435] := 0.1007951;
   t1[5436] := 0.1109563;
   t1[5437] := 0.1194762;
   t1[5438] := 0.125092;
   t1[5439] := 0.1276279;
   t1[5440] := 0.12848;
   t1[5441] := 0.129167;
   t1[5442] := 0.1312076;
   t1[5443] := 0.1361206;
   t1[5444] := 0.1449971;
   t1[5445] := 0.1386463;
   t1[5446] := 0.1128107;
   t1[5447] := 0.0913857;
   t1[5448] := 0.0779991;
   t1[5449] := 0.0714571;
   t1[5450] := 0.0688621;
   t1[5451] := 0.0673148;
   t1[5452] := 0.0639158;
   t1[5453] := 0.0558074;
   t1[5454] := 0.0422244;
   t1[5455] := 0.0254253;
   t1[5456] := 0.0079047;
   t1[5457] := -0.0078426;
   t1[5458] := -0.0193221;
   t1[5459] := -0.0244652;
   t1[5460] := -0.0415457;
   t1[5461] := -0.0350372;
   t1[5462] := -0.0175665;
   t1[5463] := 0.0128072;
   t1[5464] := 0.0534219;
   t1[5465] := 0.0999894;
   t1[5466] := 0.1482195;
   t1[5467] := 0.1938222;
   t1[5468] := 0.2325335;
   t1[5469] := 0.2613986;
   t1[5470] := 0.2793548;
   t1[5471] := 0.2854871;
   t1[5472] := 0.2788802;
   t1[5473] := 0.2586194;
   t1[5474] := 0.2243811;
   t1[5475] := -0.0568684;
   t1[5476] := -0.0272191;
   t1[5477] := 0.0124426;
   t1[5478] := 0.0640775;
   t1[5479] := 0.1232632;
   t1[5480] := 0.1833216;
   t1[5481] := 0.2375722;
   t1[5482] := 0.2793343;
   t1[5483] := 0.3020129;
   t1[5484] := 0.3032977;
   t1[5485] := 0.2870705;
   t1[5486] := 0.2576965;
   t1[5487] := 0.2195412;
   t1[5488] := 0.1769696;
   t1[5489] := 0.1340628;
   t1[5490] := -0.0039139;
   t1[5491] := 0.0191272;
   t1[5492] := 0.0457197;
   t1[5493] := 0.0756418;
   t1[5494] := 0.1067961;
   t1[5495] := 0.1364219;
   t1[5496] := 0.1617581;
   t1[5497] := 0.1800435;
   t1[5498] := 0.1885535;
   t1[5499] := 0.1863887;
   t1[5500] := 0.1752884;
   t1[5501] := 0.1571975;
   t1[5502] := 0.1340611;
   t1[5503] := 0.1078243;
   t1[5504] := 0.0803809;
   t1[5505] := 0.0001878;
   t1[5506] := -0.0121939;
   t1[5507] := -0.0135918;
   t1[5508] := -0.0001461;
   t1[5509] := 0.0261057;
   t1[5510] := 0.0610423;
   t1[5511] := 0.1005401;
   t1[5512] := 0.1404751;
   t1[5513] := 0.1767432;
   t1[5514] := 0.2062111;
   t1[5515] := 0.2271488;
   t1[5516] := 0.2379358;
   t1[5517] := 0.2369517;
   t1[5518] := 0.2225762;
   t1[5519] := 0.1939519;
   t1[5520] := 0.0901098;
   t1[5521] := 0.0856473;
   t1[5522] := 0.0847832;
   t1[5523] := 0.0890312;
   t1[5524] := 0.0971699;
   t1[5525] := 0.1070112;
   t1[5526] := 0.1163664;
   t1[5527] := 0.1230465;
   t1[5528] := 0.1248794;
   t1[5529] := 0.1205378;
   t1[5530] := 0.1099147;
   t1[5531] := 0.0929989;
   t1[5532] := 0.0697789;
   t1[5533] := 0.0402432;
   t1[5534] := 0.0047096;
   t1[5535] := 0.2602257;
   t1[5536] := 0.2587716;
   t1[5537] := 0.2539054;
   t1[5538] := 0.2456048;
   t1[5539] := 0.2350061;
   t1[5540] := 0.2236545;
   t1[5541] := 0.213096;
   t1[5542] := 0.2048765;
   t1[5543] := 0.2005251;
   t1[5544] := 0.2007389;
   t1[5545] := 0.2050117;
   t1[5546] := 0.2127433;
   t1[5547] := 0.2233339;
   t1[5548] := 0.2361833;
   t1[5549] := 0.2506394;
   t1[5550] := 0.1559216;
   t1[5551] := 0.1486253;
   t1[5552] := 0.1298461;
   t1[5553] := 0.0981546;
   t1[5554] := 0.0573184;
   t1[5555] := 0.0129418;
   t1[5556] := -0.0293689;
   t1[5557] := -0.0640073;
   t1[5558] := -0.0854428;
   t1[5559] := -0.0919368;
   t1[5560] := -0.0872303;
   t1[5561] := -0.0754922;
   t1[5562] := -0.0608914;
   t1[5563] := -0.0475969;
   t1[5564] := -0.0392405;
   t1[5565] := 0.2021459;
   t1[5566] := 0.185504;
   t1[5567] := 0.1723338;
   t1[5568] := 0.1658747;
   t1[5569] := 0.1650531;
   t1[5570] := 0.167271;
   t1[5571] := 0.1699292;
   t1[5572] := 0.1704279;
   t1[5573] := 0.1662027;
   t1[5574] := 0.1564356;
   t1[5575] := 0.1428329;
   t1[5576] := 0.1272981;
   t1[5577] := 0.1117347;
   t1[5578] := 0.0980461;
   t1[5579] := 0.0878695;
   t1[5580] := -0.0090387;
   t1[5581] := 0.0010869;
   t1[5582] := 0.0130232;
   t1[5583] := 0.0265334;
   t1[5584] := 0.0420249;
   t1[5585] := 0.0601327;
   t1[5586] := 0.0814923;
   t1[5587] := 0.1067388;
   t1[5588] := 0.1364673;
   t1[5589] := 0.169251;
   t1[5590] := 0.2007414;
   t1[5591] := 0.2263621;
   t1[5592] := 0.2415366;
   t1[5593] := 0.2416883;
   t1[5594] := 0.2231971;
   t1[5595] := 0.2351214;
   t1[5596] := 0.2108365;
   t1[5597] := 0.1878517;
   t1[5598] := 0.169596;
   t1[5599] := 0.1555034;
   t1[5600] := 0.1435958;
   t1[5601] := 0.1318934;
   t1[5602] := 0.1184166;
   t1[5603] := 0.1012091;
   t1[5604] := 0.0794922;
   t1[5605] := 0.0541886;
   t1[5606] := 0.0263538;
   t1[5607] := -0.0029565;
   t1[5608] := -0.0326869;
   t1[5609] := -0.0617994;
   t1[5610] := 0.3399203;
   t1[5611] := 0.3135424;
   t1[5612] := 0.2726368;
   t1[5613] := 0.2167182;
   t1[5614] := 0.1507169;
   t1[5615] := 0.0814768;
   t1[5616] := 0.0158441;
   t1[5617] := -0.0393348;
   t1[5618] := -0.0773026;
   t1[5619] := -0.0957355;
   t1[5620] := -0.0987177;
   t1[5621] := -0.0908337;
   t1[5622] := -0.0766682;
   t1[5623] := -0.0608055;
   t1[5624] := -0.0473261;
   t1[5625] := 0.1759748;
   t1[5626] := 0.1801888;
   t1[5627] := 0.1818157;
   t1[5628] := 0.1805558;
   t1[5629] := 0.1765932;
   t1[5630] := 0.1702829;
   t1[5631] := 0.1619801;
   t1[5632] := 0.1520399;
   t1[5633] := 0.1408151;
   t1[5634] := 0.1285303;
   t1[5635] := 0.1152255;
   t1[5636] := 0.1009261;
   t1[5637] := 0.0856576;
   t1[5638] := 0.0694454;
   t1[5639] := 0.0524179;
   t1[5640] := 0.2070498;
   t1[5641] := 0.1808508;
   t1[5642] := 0.156588;
   t1[5643] := 0.136187;
   t1[5644] := 0.1184252;
   t1[5645] := 0.1009676;
   t1[5646] := 0.0814778;
   t1[5647] := 0.0576194;
   t1[5648] := 0.0271076;
   t1[5649] := -0.009758;
   t1[5650] := -0.0489433;
   t1[5651] := -0.0861228;
   t1[5652] := -0.1169706;
   t1[5653] := -0.1371611;
   t1[5654] := -0.1431469;
   t1[5655] := 0.2326834;
   t1[5656] := 0.2043753;
   t1[5657] := 0.177029;
   t1[5658] := 0.152764;
   t1[5659] := 0.1309978;
   t1[5660] := 0.110193;
   t1[5661] := 0.0888111;
   t1[5662] := 0.0653138;
   t1[5663] := 0.0381994;
   t1[5664] := 0.0078094;
   t1[5665] := -0.0228515;
   t1[5666] := -0.0505702;
   t1[5667] := -0.072134;
   t1[5668] := -0.08433;
   t1[5669] := -0.0846053;
   t1[5670] := 0.0673334;
   t1[5671] := 0.0633753;
   t1[5672] := 0.0564422;
   t1[5673] := 0.0460167;
   t1[5674] := 0.0339294;
   t1[5675] := 0.0228404;
   t1[5676] := 0.0154107;
   t1[5677] := 0.0143013;
   t1[5678] := 0.022123;
   t1[5679] := 0.0389698;
   t1[5680] := 0.0612985;
   t1[5681] := 0.0852821;
   t1[5682] := 0.1070935;
   t1[5683] := 0.1229057;
   t1[5684] := 0.1294967;
   t1[5685] := 0.0280284;
   t1[5686] := 0.0123646;
   t1[5687] := 0.0053019;
   t1[5688] := 0.008704;
   t1[5689] := 0.02023;
   t1[5690] := 0.0360538;
   t1[5691] := 0.0523472;
   t1[5692] := 0.0652823;
   t1[5693] := 0.0710739;
   t1[5694] := 0.0680778;
   t1[5695] := 0.0577437;
   t1[5696] := 0.0417631;
   t1[5697] := 0.0218274;
   t1[5698] := -0.000372;
   t1[5699] := -0.0231627;
   t1[5700] := 0.0320975;
   t1[5701] := 0.0285746;
   t1[5702] := 0.0294266;
   t1[5703] := 0.0346239;
   t1[5704] := 0.0437935;
   t1[5705] := 0.0564409;
   t1[5706] := 0.0720719;
   t1[5707] := 0.090192;
   t1[5708] := 0.1102992;
   t1[5709] := 0.1315041;
   t1[5710] := 0.1523581;
   t1[5711] := 0.1713689;
   t1[5712] := 0.1870441;
   t1[5713] := 0.1978915;
   t1[5714] := 0.2025419;
   t1[5715] := 0.3164727;
   t1[5716] := 0.3278185;
   t1[5717] := 0.3288324;
   t1[5718] := 0.3177082;
   t1[5719] := 0.2956739;
   t1[5720] := 0.2650293;
   t1[5721] := 0.2280753;
   t1[5722] := 0.1871127;
   t1[5723] := 0.1444511;
   t1[5724] := 0.1028239;
   t1[5725] := 0.0655772;
   t1[5726] := 0.0361051;
   t1[5727] := 0.0178018;
   t1[5728] := 0.0140611;
   t1[5729] := 0.0273009;
   t1[5730] := 0.0081115;
   t1[5731] := -0.0018084;
   t1[5732] := -0.0067905;
   t1[5733] := -0.0064589;
   t1[5734] := -0.0001223;
   t1[5735] := 0.0130216;
   t1[5736] := 0.0337754;
   t1[5737] := 0.0629417;
   t1[5738] := 0.1012631;
   t1[5739] := 0.146478;
   t1[5740] := 0.1919829;
   t1[5741] := 0.2308355;
   t1[5742] := 0.2560937;
   t1[5743] := 0.260815;
   t1[5744] := 0.2395535;
   t1[5745] := 0.3116351;
   t1[5746] := 0.3089144;
   t1[5747] := 0.2948037;
   t1[5748] := 0.2666505;
   t1[5749] := 0.2263391;
   t1[5750] := 0.177357;
   t1[5751] := 0.1231935;
   t1[5752] := 0.067338;
   t1[5753] := 0.0132743;
   t1[5754] := -0.0357936;
   t1[5755] := -0.0770656;
   t1[5756] := -0.1077731;
   t1[5757] := -0.1251476;
   t1[5758] := -0.1264206;
   t1[5759] := -0.1095048;
   t1[5760] := 0.031007;
   t1[5761] := 0.0728639;
   t1[5762] := 0.1118682;
   t1[5763] := 0.1453709;
   t1[5764] := 0.1728256;
   t1[5765] := 0.1944287;
   t1[5766] := 0.2103773;
   t1[5767] := 0.2208688;
   t1[5768] := 0.226105;
   t1[5769] := 0.2265121;
   t1[5770] := 0.2228411;
   t1[5771] := 0.2158682;
   t1[5772] := 0.2063698;
   t1[5773] := 0.1951221;
   t1[5774] := 0.1828241;
   t1[5775] := -0.0120644;
   t1[5776] := 0.0343458;
   t1[5777] := 0.0716364;
   t1[5778] := 0.0958804;
   t1[5779] := 0.1085385;
   t1[5780] := 0.1129749;
   t1[5781] := 0.1125562;
   t1[5782] := 0.1106489;
   t1[5783] := 0.1105719;
   t1[5784] := 0.1132552;
   t1[5785] := 0.1161768;
   t1[5786] := 0.1165452;
   t1[5787] := 0.1115686;
   t1[5788] := 0.0984556;
   t1[5789] := 0.0751271;
   t1[5790] := 0.1167602;
   t1[5791] := 0.1561164;
   t1[5792] := 0.1873749;
   t1[5793] := 0.2071165;
   t1[5794] := 0.2158144;
   t1[5795] := 0.2153174;
   t1[5796] := 0.2074756;
   t1[5797] := 0.1941392;
   t1[5798] := 0.1771547;
   t1[5799] := 0.1581797;
   t1[5800] := 0.138599;
   t1[5801] := 0.119776;
   t1[5802] := 0.1030742;
   t1[5803] := 0.089857;
   t1[5804] := 0.0812067;
   t1[5805] := 0.2197201;
   t1[5806] := 0.2088064;
   t1[5807] := 0.1912815;
   t1[5808] := 0.1676197;
   t1[5809] := 0.1400594;
   t1[5810] := 0.1114628;
   t1[5811] := 0.0846924;
   t1[5812] := 0.0626112;
   t1[5813] := 0.0480385;
   t1[5814] := 0.0416338;
   t1[5815] := 0.0409347;
   t1[5816] := 0.0432349;
   t1[5817] := 0.0458283;
   t1[5818] := 0.0460086;
   t1[5819] := 0.0415054;
   t1[5820] := -0.0723167;
   t1[5821] := -0.0983335;
   t1[5822] := -0.1086009;
   t1[5823] := -0.1012187;
   t1[5824] := -0.0790003;
   t1[5825] := -0.0464243;
   t1[5826] := -0.0079711;
   t1[5827] := 0.0318788;
   t1[5828] := 0.0686813;
   t1[5829] := 0.0998174;
   t1[5830] := 0.1253053;
   t1[5831] := 0.1453694;
   t1[5832] := 0.1602338;
   t1[5833] := 0.1701228;
   t1[5834] := 0.1752688;
   t1[5835] := 0.0910374;
   t1[5836] := 0.1168558;
   t1[5837] := 0.1452066;
   t1[5838] := 0.1756394;
   t1[5839] := 0.2056611;
   t1[5840] := 0.2320569;
   t1[5841] := 0.2516112;
   t1[5842] := 0.2611083;
   t1[5843] := 0.2573789;
   t1[5844] := 0.239569;
   t1[5845] := 0.2101706;
   t1[5846] := 0.1719371;
   t1[5847] := 0.127622;
   t1[5848] := 0.0799786;
   t1[5849] := 0.0317715;
   t1[5850] := 0.1190348;
   t1[5851] := 0.1204072;
   t1[5852] := 0.113646;
   t1[5853] := 0.0969857;
   t1[5854] := 0.0731721;
   t1[5855] := 0.0465452;
   t1[5856] := 0.0214469;
   t1[5857] := 0.0022189;
   t1[5858] := -0.0068551;
   t1[5859] := -0.0043939;
   t1[5860] := 0.0067881;
   t1[5861] := 0.0235493;
   t1[5862] := 0.042748;
   t1[5863] := 0.0612423;
   t1[5864] := 0.0761959;
   t1[5865] := -0.0686139;
   t1[5866] := -0.0222996;
   t1[5867] := 0.0185172;
   t1[5868] := 0.0511037;
   t1[5869] := 0.0770127;
   t1[5870] := 0.0993117;
   t1[5871] := 0.1210695;
   t1[5872] := 0.1453552;
   t1[5873] := 0.1751826;
   t1[5874] := 0.210794;
   t1[5875] := 0.2484269;
   t1[5876] := 0.2840061;
   t1[5877] := 0.3134564;
   t1[5878] := 0.3327026;
   t1[5879] := 0.3382958;
   t1[5880] := -0.0348268;
   t1[5881] := -0.0604901;
   t1[5882] := -0.0801245;
   t1[5883] := -0.0922527;
   t1[5884] := -0.0973106;
   t1[5885] := -0.09641;
   t1[5886] := -0.0906634;
   t1[5887] := -0.0811834;
   t1[5888] := -0.069084;
   t1[5889] := -0.0555501;
   t1[5890] := -0.0418693;
   t1[5891] := -0.0293372;
   t1[5892] := -0.0192493;
   t1[5893] := -0.0129011;
   t1[5894] := -0.0112926;
   t1[5895] := 0.1051766;
   t1[5896] := 0.1201891;
   t1[5897] := 0.1248689;
   t1[5898] := 0.1160349;
   t1[5899] := 0.0958833;
   t1[5900] := 0.0685104;
   t1[5901] := 0.0380146;
   t1[5902] := 0.0084944;
   t1[5903] := -0.0159896;
   t1[5904] := -0.0332681;
   t1[5905] := -0.0439053;
   t1[5906] := -0.0486786;
   t1[5907] := -0.0483656;
   t1[5908] := -0.0437438;
   t1[5909] := -0.0355984;
   t1[5910] := 0.117127;
   t1[5911] := 0.1148726;
   t1[5912] := 0.111075;
   t1[5913] := 0.1054802;
   t1[5914] := 0.0976384;
   t1[5915] := 0.0870302;
   t1[5916] := 0.0731363;
   t1[5917] := 0.0554375;
   t1[5918] := 0.033439;
   t1[5919] := 0.007884;
   t1[5920] := -0.0186958;
   t1[5921] := -0.0436292;
   t1[5922] := -0.0642449;
   t1[5923] := -0.0778715;
   t1[5924] := -0.0823112;
   t1[5925] := 0.0605384;
   t1[5926] := 0.0586405;
   t1[5927] := 0.0612945;
   t1[5928] := 0.0696282;
   t1[5929] := 0.081501;
   t1[5930] := 0.093617;
   t1[5931] := 0.1026793;
   t1[5932] := 0.1053907;
   t1[5933] := 0.0985063;
   t1[5934] := 0.0813848;
   t1[5935] := 0.0571482;
   t1[5936] := 0.0292125;
   t1[5937] := 0.0009933;
   t1[5938] := -0.0240935;
   t1[5939] := -0.0430221;
   t1[5940] := 0.0497248;
   t1[5941] := 0.0665747;
   t1[5942] := 0.0795811;
   t1[5943] := 0.0878671;
   t1[5944] := 0.0923519;
   t1[5945] := 0.0945895;
   t1[5946] := 0.0961348;
   t1[5947] := 0.0985424;
   t1[5948] := 0.1033362;
   t1[5949] := 0.1104933;
   t1[5950] := 0.1177552;
   t1[5951] := 0.1226891;
   t1[5952] := 0.122862;
   t1[5953] := 0.1158412;
   t1[5954] := 0.0997852;
   t1[5955] := 0.1509402;
   t1[5956] := 0.1378048;
   t1[5957] := 0.1266288;
   t1[5958] := 0.1189594;
   t1[5959] := 0.1148499;
   t1[5960] := 0.1138258;
   t1[5961] := 0.1154119;
   t1[5962] := 0.119133;
   t1[5963] := 0.124502;
   t1[5964] := 0.1304314;
   t1[5965] := 0.134966;
   t1[5966] := 0.1360831;
   t1[5967] := 0.1317597;
   t1[5968] := 0.1199732;
   t1[5969] := 0.0993125;
   t1[5970] := 0.1816427;
   t1[5971] := 0.1953361;
   t1[5972] := 0.2048154;
   t1[5973] := 0.2091279;
   t1[5974] := 0.2077178;
   t1[5975] := 0.2001692;
   t1[5976] := 0.1860666;
   t1[5977] := 0.1649944;
   t1[5978] := 0.1365594;
   t1[5979] := 0.1014875;
   t1[5980] := 0.0621217;
   t1[5981] := 0.0209314;
   t1[5982] := -0.0196139;
   t1[5983] := -0.0570451;
   t1[5984] := -0.089056;
   t1[5985] := 0.0638854;
   t1[5986] := 0.0921957;
   t1[5987] := 0.1206934;
   t1[5988] := 0.1466806;
   t1[5989] := 0.1683184;
   t1[5990] := 0.1840713;
   t1[5991] := 0.1924042;
   t1[5992] := 0.1917821;
   t1[5993] := 0.1807017;
   t1[5994] := 0.1592482;
   t1[5995] := 0.1298026;
   t1[5996] := 0.0949252;
   t1[5997] := 0.0571763;
   t1[5998] := 0.019116;
   t1[5999] := -0.0168727;
   t1[6000] := -0.0008921;
   t1[6001] := -0.003162;
   t1[6002] := 0.0025781;
   t1[6003] := 0.0173504;
   t1[6004] := 0.0402556;
   t1[6005] := 0.0697151;
   t1[6006] := 0.1041497;
   t1[6007] := 0.1419802;
   t1[6008] := 0.1816104;
   t1[6009] := 0.2206014;
   t1[6010] := 0.2552963;
   t1[6011] := 0.2819431;
   t1[6012] := 0.2967896;
   t1[6013] := 0.2960841;
   t1[6014] := 0.2769434;
   t1[6015] := 0.1006214;
   t1[6016] := 0.0653474;
   t1[6017] := 0.0373836;
   t1[6018] := 0.0202273;
   t1[6019] := 0.0144889;
   t1[6020] := 0.0197586;
   t1[6021] := 0.0356257;
   t1[6022] := 0.0616793;
   t1[6023] := 0.0974702;
   t1[6024] := 0.1406413;
   t1[6025] := 0.186077;
   t1[6026] := 0.2284468;
   t1[6027] := 0.2624199;
   t1[6028] := 0.2826659;
   t1[6029] := 0.2847723;
   t1[6030] := 0.0050532;
   t1[6031] := 0.0100576;
   t1[6032] := 0.0124636;
   t1[6033] := 0.0122359;
   t1[6034] := 0.0100102;
   t1[6035] := 0.0066595;
   t1[6036] := 0.003057;
   t1[6037] := 7.58E-05;
   t1[6038] := -0.0014203;
   t1[6039] := -0.0010509;
   t1[6040] := 0.0008668;
   t1[6041] := 0.0039609;
   t1[6042] := 0.0078595;
   t1[6043] := 0.0121909;
   t1[6044] := 0.0165797;
   t1[6045] := 0.1193422;
   t1[6046] := 0.1024935;
   t1[6047] := 0.0896988;
   t1[6048] := 0.0821659;
   t1[6049] := 0.0787474;
   t1[6050] := 0.0774642;
   t1[6051] := 0.0763359;
   t1[6052] := 0.0733823;
   t1[6053] := 0.0666513;
   t1[6054] := 0.0556094;
   t1[6055] := 0.0417721;
   t1[6056] := 0.0268153;
   t1[6057] := 0.0124147;
   t1[6058] := 0.0002461;
   t1[6059] := -0.0082943;
   t1[6060] := 0.1559757;
   t1[6061] := 0.1248735;
   t1[6062] := 0.0970409;
   t1[6063] := 0.0750365;
   t1[6064] := 0.0575972;
   t1[6065] := 0.0421093;
   t1[6066] := 0.0259577;
   t1[6067] := 0.0065271;
   t1[6068] := -0.0187525;
   t1[6069] := -0.0501943;
   t1[6070] := -0.0848498;
   t1[6071] := -0.1195156;
   t1[6072] := -0.1509886;
   t1[6073] := -0.1760656;
   t1[6074] := -0.1919876;
   t1[6075] := 0.0302589;
   t1[6076] := 0.0111427;
   t1[6077] := 0.001131;
   t1[6078] := 0.0024504;
   t1[6079] := 0.0129941;
   t1[6080] := 0.0291245;
   t1[6081] := 0.047202;
   t1[6082] := 0.063587;
   t1[6083] := 0.0746798;
   t1[6084] := 0.0788727;
   t1[6085] := 0.0774371;
   t1[6086] := 0.0718691;
   t1[6087] := 0.0636648;
   t1[6088] := 0.0543203;
   t1[6089] := 0.0451873;
   t1[6090] := -0.0808457;
   t1[6091] := -0.0954091;
   t1[6092] := -0.101415;
   t1[6093] := -0.0956159;
   t1[6094] := -0.0797668;
   t1[6095] := -0.0573905;
   t1[6096] := -0.0320114;
   t1[6097] := -0.0071543;
   t1[6098] := 0.013699;
   t1[6099] := 0.0292106;
   t1[6100] := 0.0411408;
   t1[6101] := 0.051492;
   t1[6102] := 0.0622665;
   t1[6103] := 0.0754664;
   t1[6104] := 0.0926117;
   t1[6105] := 0.2293762;
   t1[6106] := 0.2092099;
   t1[6107] := 0.1841759;
   t1[6108] := 0.1542055;
   t1[6109] := 0.1199331;
   t1[6110] := 0.0822419;
   t1[6111] := 0.0420152;
   t1[6112] := 0.0001365;
   t1[6113] := -0.0425065;
   t1[6114] := -0.0848117;
   t1[6115] := -0.1253664;
   t1[6116] := -0.162734;
   t1[6117] := -0.1954777;
   t1[6118] := -0.2221611;
   t1[6119] := -0.2415285;
   t1[6120] := -0.0665781;
   t1[6121] := -0.0948688;
   t1[6122] := -0.110597;
   t1[6123] := -0.1103839;
   t1[6124] := -0.0966698;
   t1[6125] := -0.0739512;
   t1[6126] := -0.046727;
   t1[6127] := -0.0194959;
   t1[6128] := 0.0032941;
   t1[6129] := 0.0197511;
   t1[6130] := 0.0316765;
   t1[6131] := 0.0411602;
   t1[6132] := 0.0502922;
   t1[6133] := 0.0611624;
   t1[6134] := 0.0753623;
   t1[6135] := -0.2079995;
   t1[6136] := -0.2293701;
   t1[6137] := -0.2417559;
   t1[6138] := -0.2408475;
   t1[6139] := -0.226425;
   t1[6140] := -0.1997138;
   t1[6141] := -0.1619405;
   t1[6142] := -0.1143323;
   t1[6143] := -0.0581369;
   t1[6144] := 0.0043453;
   t1[6145] := 0.0692932;
   t1[6146] := 0.1327671;
   t1[6147] := 0.190827;
   t1[6148] := 0.2395333;
   t1[6149] := 0.2753775;
   t1[6150] := 0.1881377;
   t1[6151] := 0.1954438;
   t1[6152] := 0.1860857;
   t1[6153] := 0.1549516;
   t1[6154] := 0.1066808;
   t1[6155] := 0.0493579;
   t1[6156] := -0.0089286;
   t1[6157] := -0.0600901;
   t1[6158] := -0.0961361;
   t1[6159] := -0.1139835;
   t1[6160] := -0.1176418;
   t1[6161] := -0.1116738;
   t1[6162] := -0.1006425;
   t1[6163] := -0.089111;
   t1[6164] := -0.08102;
   t1[6165] := 0.3099137;
   t1[6166] := 0.3089272;
   t1[6167] := 0.2974539;
   t1[6168] := 0.2727434;
   t1[6169] := 0.2367496;
   t1[6170] := 0.193089;
   t1[6171] := 0.14538;
   t1[6172] := 0.0972409;
   t1[6173] := 0.0522519;
   t1[6174] := 0.0120826;
   t1[6175] := -0.0243583;
   t1[6176] := -0.058378;
   t1[6177] := -0.0912833;
   t1[6178] := -0.1243813;
   t1[6179] := -0.1586504;
   t1[6180] := -0.1184668;
   t1[6181] := -0.1011787;
   t1[6182] := -0.0832939;
   t1[6183] := -0.065112;
   t1[6184] := -0.0449892;
   t1[6185] := -0.0205951;
   t1[6186] := 0.0104014;
   t1[6187] := 0.0503315;
   t1[6188] := 0.1014512;
   t1[6189] := 0.162256;
   t1[6190] := 0.2258063;
   t1[6191] := 0.2847385;
   t1[6192] := 0.3316885;
   t1[6193] := 0.3592928;
   t1[6194] := 0.3615301;
   t1[6195] := -0.091948;
   t1[6196] := -0.0989024;
   t1[6197] := -0.0981292;
   t1[6198] := -0.0886809;
   t1[6199] := -0.0724812;
   t1[6200] := -0.0524682;
   t1[6201] := -0.0315812;
   t1[6202] := -0.0127595;
   t1[6203] := 0.0011018;
   t1[6204] := 0.009312;
   t1[6205] := 0.0143668;
   t1[6206] := 0.0190103;
   t1[6207] := 0.0259871;
   t1[6208] := 0.0380413;
   t1[6209] := 0.0572519;
   t1[6210] := -0.0519979;
   t1[6211] := -0.0109861;
   t1[6212] := 0.0238115;
   t1[6213] := 0.0496663;
   t1[6214] := 0.0678337;
   t1[6215] := 0.0809767;
   t1[6216] := 0.09176;
   t1[6217] := 0.1028482;
   t1[6218] := 0.1168682;
   t1[6219] := 0.1345674;
   t1[6220] := 0.1539759;
   t1[6221] := 0.1729119;
   t1[6222] := 0.1891934;
   t1[6223] := 0.2006386;
   t1[6224] := 0.2053535;
   t1[6225] := 0.0139801;
   t1[6226] := 0.0765099;
   t1[6227] := 0.124489;
   t1[6228] := 0.1503144;
   t1[6229] := 0.1560223;
   t1[6230] := 0.1470548;
   t1[6231] := 0.128858;
   t1[6232] := 0.1068778;
   t1[6233] := 0.0865192;
   t1[6234] := 0.0711201;
   t1[6235] := 0.0610319;
   t1[6236] := 0.056373;
   t1[6237] := 0.0572614;
   t1[6238] := 0.0638156;
   t1[6239] := 0.0758494;
   t1[6240] := -0.0209548;
   t1[6241] := -0.0179487;
   t1[6242] := -0.0127916;
   t1[6243] := -0.0054356;
   t1[6244] := 0.0040806;
   t1[6245] := 0.0156877;
   t1[6246] := 0.0293165;
   t1[6247] := 0.0448978;
   t1[6248] := 0.0623495;
   t1[6249] := 0.0809498;
   t1[6250] := 0.0990518;
   t1[6251] := 0.1149368;
   t1[6252] := 0.1268858;
   t1[6253] := 0.1331799;
   t1[6254] := 0.1324356;
   t1[6255] := -0.1402293;
   t1[6256] := -0.0966064;
   t1[6257] := -0.0542916;
   t1[6258] := -0.0159849;
   t1[6259] := 0.0178334;
   t1[6260] := 0.0474672;
   t1[6261] := 0.0732214;
   t1[6262] := 0.0954007;
   t1[6263] := 0.1143034;
   t1[6264] := 0.1298921;
   t1[6265] := 0.1416449;
   t1[6266] := 0.1490018;
   t1[6267] := 0.1514029;
   t1[6268] := 0.1482883;
   t1[6269] := 0.1393104;
   t1[6270] := -0.0203112;
   t1[6271] := 0.0038462;
   t1[6272] := 0.0274046;
   t1[6273] := 0.0485846;
   t1[6274] := 0.0672529;
   t1[6275] := 0.0838573;
   t1[6276] := 0.0988465;
   t1[6277] := 0.1126692;
   t1[6278] := 0.1257661;
   t1[6279] := 0.1381858;
   t1[6280] := 0.1494099;
   t1[6281] := 0.1588758;
   t1[6282] := 0.1660208;
   t1[6283] := 0.1702823;
   t1[6284] := 0.171152;
   t1[6285] := 0.046874;
   t1[6286] := 0.0112669;
   t1[6287] := -0.0174814;
   t1[6288] := -0.0371403;
   t1[6289] := -0.0470314;
   t1[6290] := -0.0470243;
   t1[6291] := -0.0369892;
   t1[6292] := -0.0167964;
   t1[6293] := 0.0136476;
   t1[6294] := 0.0526369;
   t1[6295] := 0.0958637;
   t1[6296] := 0.1388175;
   t1[6297] := 0.1769875;
   t1[6298] := 0.2058632;
   t1[6299] := 0.2215942;
   t1[6300] := -0.0061098;
   t1[6301] := -0.0204832;
   t1[6302] := -0.0380719;
   t1[6303] := -0.0586594;
   t1[6304] := -0.0799497;
   t1[6305] := -0.0989121;
   t1[6306] := -0.1125149;
   t1[6307] := -0.1177266;
   t1[6308] := -0.1115672;
   t1[6309] := -0.0936386;
   t1[6310] := -0.0672741;
   t1[6311] := -0.0360984;
   t1[6312] := -0.0037362;
   t1[6313] := 0.0261879;
   t1[6314] := 0.0504587;
   t1[6315] := 0.0525412;
   t1[6316] := 0.0487455;
   t1[6317] := 0.0483423;
   t1[6318] := 0.0520326;
   t1[6319] := 0.0593908;
   t1[6320] := 0.0695932;
   t1[6321] := 0.0818158;
   t1[6322] := 0.0952343;
   t1[6323] := 0.109027;
   t1[6324] := 0.1224888;
   t1[6325] := 0.1350833;
   t1[6326] := 0.1462873;
   t1[6327] := 0.1555775;
   t1[6328] := 0.1624307;
   t1[6329] := 0.1664159;
   t1[6330] := 0.0825259;
   t1[6331] := 0.0992742;
   t1[6332] := 0.1090136;
   t1[6333] := 0.1097467;
   t1[6334] := 0.1029049;
   t1[6335] := 0.0911318;
   t1[6336] := 0.0770722;
   t1[6337] := 0.0633709;
   t1[6338] := 0.0526507;
   t1[6339] := 0.0464374;
   t1[6340] := 0.0446709;
   t1[6341] := 0.0471674;
   t1[6342] := 0.0537429;
   t1[6343] := 0.0642136;
   t1[6344] := 0.0782398;
   t1[6345] := 0.1141067;
   t1[6346] := 0.1003176;
   t1[6347] := 0.092636;
   t1[6348] := 0.0935227;
   t1[6349] := 0.1012303;
   t1[6350] := 0.1125243;
   t1[6351] := 0.1241685;
   t1[6352] := 0.1329268;
   t1[6353] := 0.1355985;
   t1[6354] := 0.1307586;
   t1[6355] := 0.1195484;
   t1[6356] := 0.1033096;
   t1[6357] := 0.0833837;
   t1[6358] := 0.0611126;
   t1[6359] := 0.0378071;
   t1[6360] := -0.0047682;
   t1[6361] := 0.0300573;
   t1[6362] := 0.0613615;
   t1[6363] := 0.0850331;
   t1[6364] := 0.1001842;
   t1[6365] := 0.107066;
   t1[6366] := 0.1059313;
   t1[6367] := 0.0970326;
   t1[6368] := 0.0806607;
   t1[6369] := 0.0590239;
   t1[6370] := 0.0371009;
   t1[6371] := 0.0200866;
   t1[6372] := 0.0131764;
   t1[6373] := 0.0215651;
   t1[6374] := 0.0493127;
   t1[6375] := -0.0994751;
   t1[6376] := -0.0872729;
   t1[6377] := -0.0710769;
   t1[6378] := -0.0517855;
   t1[6379] := -0.031381;
   t1[6380] := -0.0122285;
   t1[6381] := 0.0033061;
   t1[6382] := 0.0128573;
   t1[6383] := 0.014107;
   t1[6384] := 0.0071194;
   t1[6385] := -0.0045978;
   t1[6386] := -0.0172684;
   t1[6387] := -0.027116;
   t1[6388] := -0.0303644;
   t1[6389] := -0.0240877;
   t1[6390] := -0.0279364;
   t1[6391] := -0.0443435;
   t1[6392] := -0.0566576;
   t1[6393] := -0.0631468;
   t1[6394] := -0.0632291;
   t1[6395] := -0.0567285;
   t1[6396] := -0.0434695;
   t1[6397] := -0.0232766;
   t1[6398] := 0.0040068;
   t1[6399] := 0.0376029;
   t1[6400] := 0.0753821;
   t1[6401] := 0.1151099;
   t1[6402] := 0.1545514;
   t1[6403] := 0.191472;
   t1[6404] := 0.2237596;
   t1[6405] := -0.0601228;
   t1[6406] := -0.0832199;
   t1[6407] := -0.0936729;
   t1[6408] := -0.0874911;
   t1[6409] := -0.0672874;
   t1[6410] := -0.038008;
   t1[6411] := -0.0046016;
   t1[6412] := 0.0279829;
   t1[6413] := 0.0548454;
   t1[6414] := 0.0735277;
   t1[6415] := 0.0851004;
   t1[6416] := 0.0909095;
   t1[6417] := 0.0923011;
   t1[6418] := 0.0906214;
   t1[6419] := 0.0871147;
   t1[6420] := -0.0200038;
   t1[6421] := -0.0350584;
   t1[6422] := -0.0439363;
   t1[6423] := -0.044188;
   t1[6424] := -0.0373529;
   t1[6425] := -0.0263804;
   t1[6426] := -0.0142212;
   t1[6427] := -0.0038263;
   t1[6428] := 0.0018905;
   t1[6429] := 0.001859;
   t1[6430] := -0.0023258;
   t1[6431] := -0.008861;
   t1[6432] := -0.0159436;
   t1[6433] := -0.0217707;
   t1[6434] := -0.0247319;
   t1[6435] := 0.0827025;
   t1[6436] := 0.0827253;
   t1[6437] := 0.082019;
   t1[6438] := 0.0818175;
   t1[6439] := 0.0826003;
   t1[6440] := 0.0845807;
   t1[6441] := 0.0879711;
   t1[6442] := 0.0929846;
   t1[6443] := 0.0998287;
   t1[6444] := 0.1084578;
   t1[6445] := 0.1184602;
   t1[6446] := 0.1293955;
   t1[6447] := 0.1408234;
   t1[6448] := 0.1523036;
   t1[6449] := 0.163317;
   t1[6450] := -0.2512962;
   t1[6451] := -0.2215711;
   t1[6452] := -0.1824992;
   t1[6453] := -0.1332904;
   t1[6454] := -0.0765017;
   t1[6455] := -0.0158731;
   t1[6456] := 0.0448542;
   t1[6457] := 0.1019388;
   t1[6458] := 0.1516734;
   t1[6459] := 0.1920538;
   t1[6460] := 0.2235361;
   t1[6461] := 0.2467691;
   t1[6462] := 0.2624012;
   t1[6463] := 0.2710811;
   t1[6464] := 0.2734145;
   t1[6465] := -0.1341166;
   t1[6466] := -0.1159058;
   t1[6467] := -0.0960976;
   t1[6468] := -0.0760673;
   t1[6469] := -0.0554031;
   t1[6470] := -0.0330623;
   t1[6471] := -0.0080015;
   t1[6472] := 0.0208229;
   t1[6473] := 0.0544231;
   t1[6474] := 0.0922494;
   t1[6475] := 0.1314942;
   t1[6476] := 0.1691739;
   t1[6477] := 0.2023047;
   t1[6478] := 0.227903;
   t1[6479] := 0.2433818;
   t1[6480] := -0.1029919;
   t1[6481] := -0.0621915;
   t1[6482] := -0.0279917;
   t1[6483] := -0.0040313;
   t1[6484] := 0.0097049;
   t1[6485] := 0.0145226;
   t1[6486] := 0.0117293;
   t1[6487] := 0.0026323;
   t1[6488] := -0.0114623;
   t1[6489] := -0.0293128;
   t1[6490] := -0.0497706;
   t1[6491] := -0.0716944;
   t1[6492] := -0.093943;
   t1[6493] := -0.1153751;
   t1[6494] := -0.1348667;
   t1[6495] := -0.0090596;
   t1[6496] := 0.0081976;
   t1[6497] := 0.017534;
   t1[6498] := 0.0162086;
   t1[6499] := 0.0063039;
   t1[6500] := -0.0083936;
   t1[6501] := -0.0240951;
   t1[6502] := -0.0370122;
   t1[6503] := -0.0434054;
   t1[6504] := -0.0420007;
   t1[6505] := -0.0350874;
   t1[6506] := -0.0252325;
   t1[6507] := -0.0150034;
   t1[6508] := -0.0069672;
   t1[6509] := -0.0033141;
   t1[6510] := -0.192581;
   t1[6511] := -0.1531844;
   t1[6512] := -0.1149055;
   t1[6513] := -0.0804899;
   t1[6514] := -0.0505305;
   t1[6515] := -0.0248594;
   t1[6516] := -0.003308;
   t1[6517] := 0.0142924;
   t1[6518] := 0.0281083;
   t1[6519] := 0.0382035;
   t1[6520] := 0.0444928;
   t1[6521] := 0.0468797;
   t1[6522] := 0.0452672;
   t1[6523] := 0.0395589;
   t1[6524] := 0.0298061;
   t1[6525] := 0.1197442;
   t1[6526] := 0.1433934;
   t1[6527] := 0.1682112;
   t1[6528] := 0.1935416;
   t1[6529] := 0.2158445;
   t1[6530] := 0.2305607;
   t1[6531] := 0.2331294;
   t1[6532] := 0.2189904;
   t1[6533] := 0.1836909;
   t1[6534] := 0.1281663;
   t1[6535] := 0.0611394;
   t1[6536] := -0.0080591;
   t1[6537] := -0.0700983;
   t1[6538] := -0.1156476;
   t1[6539] := -0.1369247;
   t1[6540] := 0.1101966;
   t1[6541] := 0.090723;
   t1[6542] := 0.0662378;
   t1[6543] := 0.0375331;
   t1[6544] := 0.0052269;
   t1[6545] := -0.0301243;
   t1[6546] := -0.0679642;
   t1[6547] := -0.1077363;
   t1[6548] := -0.1488545;
   t1[6549] := -0.1892368;
   t1[6550] := -0.2246395;
   t1[6551] := -0.2506505;
   t1[6552] := -0.2628575;
   t1[6553] := -0.2568482;
   t1[6554] := -0.2293048;
   t1[6555] := -0.2120533;
   t1[6556] := -0.1725074;
   t1[6557] := -0.1343032;
   t1[6558] := -0.10056;
   t1[6559] := -0.0706636;
   t1[6560] := -0.0426809;
   t1[6561] := -0.0146768;
   t1[6562] := 0.0152835;
   t1[6563] := 0.0490809;
   t1[6564] := 0.0859011;
   t1[6565] := 0.1210342;
   t1[6566] := 0.1494662;
   t1[6567] := 0.1661831;
   t1[6568] := 0.166171;
   t1[6569] := 0.1456208;
   t1[6570] := 0.0065645;
   t1[6571] := 0.0255592;
   t1[6572] := 0.0313356;
   t1[6573] := 0.0210245;
   t1[6574] := -0.001631;
   t1[6575] := -0.0305509;
   t1[6576] := -0.0596525;
   t1[6577] := -0.0828533;
   t1[6578] := -0.0941494;
   t1[6579] := -0.091473;
   t1[6580] := -0.0784451;
   t1[6581] := -0.0591306;
   t1[6582] := -0.0375945;
   t1[6583] := -0.0179019;
   t1[6584] := -0.0036363;
   t1[6585] := -0.1478585;
   t1[6586] := -0.1016801;
   t1[6587] := -0.0534096;
   t1[6588] := -0.0045012;
   t1[6589] := 0.0430296;
   t1[6590] := 0.0869689;
   t1[6591] := 0.1251023;
   t1[6592] := 0.1552157;
   t1[6593] := 0.1751249;
   t1[6594] := 0.1841438;
   t1[6595] := 0.1837518;
   t1[6596] := 0.1755973;
   t1[6597] := 0.1613284;
   t1[6598] := 0.1425938;
   t1[6599] := 0.1209146;
   t1[6600] := 0.1370825;
   t1[6601] := 0.1420729;
   t1[6602] := 0.1393185;
   t1[6603] := 0.1268324;
   t1[6604] := 0.1072708;
   t1[6605] := 0.0849311;
   t1[6606] := 0.064112;
   t1[6607] := 0.0491126;
   t1[6608] := 0.044159;
   t1[6609] := 0.0498348;
   t1[6610] := 0.0614587;
   t1[6611] := 0.0739385;
   t1[6612] := 0.0821821;
   t1[6613] := 0.0810973;
   t1[6614] := 0.0665991;
   t1[6615] := 0.1807702;
   t1[6616] := 0.1565812;
   t1[6617] := 0.130707;
   t1[6618] := 0.1046203;
   t1[6619] := 0.0797492;
   t1[6620] := 0.0575057;
   t1[6621] := 0.0393019;
   t1[6622] := 0.0265498;
   t1[6623] := 0.0206299;
   t1[6624] := 0.021339;
   t1[6625] := 0.0261853;
   t1[6626] := 0.0324982;
   t1[6627] := 0.0376073;
   t1[6628] := 0.0388422;
   t1[6629] := 0.0340154;
   t1[6630] := 0.1694753;
   t1[6631] := 0.1208992;
   t1[6632] := 0.0777849;
   t1[6633] := 0.0448265;
   t1[6634] := 0.0206269;
   t1[6635] := 0.0016371;
   t1[6636] := -0.015695;
   t1[6637] := -0.0349208;
   t1[6638] := -0.0595318;
   t1[6639] := -0.0899906;
   t1[6640] := -0.1223832;
   t1[6641] := -0.1524539;
   t1[6642] := -0.1759469;
   t1[6643] := -0.1886065;
   t1[6644] := -0.1869699;
   t1[6645] := 0.1395302;
   t1[6646] := 0.1353829;
   t1[6647] := 0.1285779;
   t1[6648] := 0.1179194;
   t1[6649] := 0.1044381;
   t1[6650] := 0.0899512;
   t1[6651] := 0.0762769;
   t1[6652] := 0.0652332;
   t1[6653] := 0.0586142;
   t1[6654] := 0.0569994;
   t1[6655] := 0.0592136;
   t1[6656] := 0.0639448;
   t1[6657] := 0.0698806;
   t1[6658] := 0.0757091;
   t1[6659] := 0.0802208;
   t1[6660] := 0.1470823;
   t1[6661] := 0.1179306;
   t1[6662] := 0.0816353;
   t1[6663] := 0.0405737;
   t1[6664] := -0.0027442;
   t1[6665] := -0.0457612;
   t1[6666] := -0.0859203;
   t1[6667] := -0.1206642;
   t1[6668] := -0.1474703;
   t1[6669] := -0.165546;
   t1[6670] := -0.1765982;
   t1[6671] := -0.1825293;
   t1[6672] := -0.1852415;
   t1[6673] := -0.1866371;
   t1[6674] := -0.1882973;
   t1[6675] := 0.2214328;
   t1[6676] := 0.167643;
   t1[6677] := 0.1152031;
   t1[6678] := 0.0675413;
   t1[6679] := 0.0258469;
   t1[6680] := -0.0094813;
   t1[6681] := -0.0380455;
   t1[6682] := -0.059448;
   t1[6683] := -0.0733068;
   t1[6684] := -0.0800316;
   t1[6685] := -0.081176;
   t1[6686] := -0.0783831;
   t1[6687] := -0.0732959;
   t1[6688] := -0.0675574;
   t1[6689] := -0.0626088;
   t1[6690] := 0.123815;
   t1[6691] := 0.1223871;
   t1[6692] := 0.1153592;
   t1[6693] := 0.1030973;
   t1[6694] := 0.0870451;
   t1[6695] := 0.0690272;
   t1[6696] := 0.0508686;
   t1[6697] := 0.0343944;
   t1[6698] := 0.0214091;
   t1[6699] := 0.0126934;
   t1[6700] := 0.007548;
   t1[6701] := 0.0051582;
   t1[6702] := 0.0047093;
   t1[6703] := 0.0053864;
   t1[6704] := 0.0064445;
   t1[6705] := 0.3236379;
   t1[6706] := 0.2845902;
   t1[6707] := 0.2380731;
   t1[6708] := 0.185373;
   t1[6709] := 0.1287298;
   t1[6710] := 0.0707202;
   t1[6711] := 0.0139215;
   t1[6712] := -0.0390891;
   t1[6713] := -0.0857643;
   t1[6714] := -0.125057;
   t1[6715] := -0.1580877;
   t1[6716] := -0.1861463;
   t1[6717] := -0.2105227;
   t1[6718] := -0.2325067;
   t1[6719] := -0.2530213;
   w2[0] := 0.3822261;
   w2[1] := 0.6735258;
   w2[2] := 0.4999258;
   w2[3] := 0.0709843;
   w2[4] := 0.4040336;
   w2[5] := -0.3168498;
   w2[6] := -0.5318553;
   w2[7] := -0.3348889;
   w2[8] := 0.5234552;
   w2[9] := 0.3241403;
   w2[10] := -0.6014917;
   w2[11] := -0.2869324;
   w2[12] := -0.0813316;
   w2[13] := 0.2735443;
   w2[14] := -0.5975453;
   w2[15] := -0.3671676;
   w2[16] := 0.1604395;
   w2[17] := 0.6218057;
   w2[18] := -0.535407;
   w2[19] := -0.428839;
   w2[20] := 0.4432988;
   w2[21] := -0.1195226;
   w2[22] := -0.1593684;
   w2[23] := -0.4208567;
   w2[24] := -0.0164311;
   w2[25] := 0.1177106;
   w2[26] := -0.1915699;
   w2[27] := -0.2585908;
   w2[28] := 0.7388805;
   w2[29] := 0.7177937;
   w2[30] := 0.9066412;
   w2[31] := -0.3313666;
   w2[32] := -0.5566195;
   w2[33] := 0.1009696;
   w2[34] := 0.7024983;
   w2[35] := -0.0061407;
   w2[36] := 0.9221094;
   w2[37] := 0.9728315;
   w2[38] := 0.7287791;
   w2[39] := 0.1011917;
   w2[40] := 0.1708561;
   w2[41] := 0.0181266;
   w2[42] := -0.3799455;
   w2[43] := -0.2221509;
   w2[44] := -0.2996568;
   w2[45] := 0.1856399;
   w2[46] := -0.2363337;
   w2[47] := 0.3469633;
   w2[48] := -0.3170906;
   w2[49] := -0.3010724;
   w2[50] := -0.4463713;
   w2[51] := 0.4818622;
   w2[52] := -0.2695292;
   w2[53] := -0.4620254;
   w2[54] := 0.0533027;
   w2[55] := -0.395156;
   w2[56] := 0.0408355;
   w2[57] := -0.2507218;
   w2[58] := 0.0280879;
   w2[59] := 0.0458854;
   w2[60] := -0.0139494;
   w2[61] := 0.0098419;
   w2[62] := -0.4868755;
   w2[63] := 0.1032088;
   w2[64] := 0.1231787;
   w2[65] := 0.5223995;
   w2[66] := 0.4042619;
   w2[67] := 0.2341684;
   w2[68] := -0.2304757;
   w2[69] := 0.0635033;
   w2[70] := -0.3774453;
   w2[71] := -0.4428134;
   w2[72] := -0.0484126;
   w2[73] := 0.2895669;
   w2[74] := -0.6764416;
   w2[75] := -0.3088431;
   w2[76] := 0.4827037;
   w2[77] := 0.0691548;
   w2[78] := 0.4661854;
   w2[79] := 0.1204736;
   w2[80] := -0.4872637;
   w2[81] := -0.0951735;
   w2[82] := -0.0189593;
   w2[83] := -0.1372051;
   w2[84] := -0.9140335;
   w2[85] := -0.8600995;
   w2[86] := -1.056187;
   w2[87] := -0.5128109;
   w2[88] := -0.7898985;
   w2[89] := -0.5083115;
   w2[90] := -0.5282256;
   w2[91] := -0.4263123;
   w2[92] := -1.016044;
   w2[93] := -0.0212463;
   w2[94] := 0.6550046;
   w2[95] := 0.4706961;
   w2[96] := -0.1141442;
   w2[97] := -0.2175039;
   w2[98] := -0.2840221;
   w2[99] := -0.3306261;
   w2[100] := -0.2441688;
   w2[101] := 0.3605514;
   w2[102] := -0.3955784;
   w2[103] := 0.0529358;
   w2[104] := 0.3398173;
   w2[105] := 0.3715278;
   w2[106] := 0.429172;
   w2[107] := 0.4002611;
   w2[108] := -0.2264336;
   w2[109] := 0.312763;
   w2[110] := 0.5647593;
   w2[111] := 0.0224205;
   w2[112] := -0.5216327;
   w2[113] := -0.2093005;
   w2[114] := -0.3824884;
   w2[115] := -0.0496232;
   w2[116] := -0.0204715;
   w2[117] := 0.3446302;
   w2[118] := -0.1566623;
   w2[119] := -0.1314349;
   w2[120] := -0.3364701;
   w2[121] := -0.5365704;
   w2[122] := -0.3706124;
   w2[123] := -0.2384351;
   w2[124] := 0.2599077;
   w2[125] := 0.0878742;
   w2[126] := -0.1167608;
   w2[127] := 0.4445257;
   w2[128] := 0.0472859;
   w2[129] := -0.2039315;
   w2[130] := -0.0123044;
   w2[131] := 0.5347427;
   w2[132] := -0.4565654;
   w2[133] := -0.1309683;
   w2[134] := -0.1916631;
   w2[135] := -0.0229556;
   w2[136] := -0.1463313;
   w2[137] := 0.0884493;
   w2[138] := -0.1268248;
   w2[139] := 0.1727386;
   w2[140] := 0.1864566;
   w2[141] := 0.0450289;
   w2[142] := 0.2544484;
   w2[143] := -0.1416016;
   w2[144] := -0.1781151;
   w2[145] := -0.1914191;
   w2[146] := 0.3022377;
   w2[147] := 0.2656204;
   w2[148] := 0.135544;
   w2[149] := 0.5225624;
   w2[150] := 0.8165789;
   w2[151] := 0.3793563;
   w2[152] := -0.1251971;
   w2[153] := -0.032513;
   w2[154] := -0.1753309;
   w2[155] := -0.429324;
   w2[156] := -0.4619711;
   w2[157] := 0.3961401;
   w2[158] := -0.6358346;
   w2[159] := 0.531637;
   w2[160] := 0.2908633;
   w2[161] := 0.2183272;
   w2[162] := 0.3942987;
   w2[163] := 0.3020125;
   w2[164] := -0.4793546;
   w2[165] := 0.0537859;
   w2[166] := 0.2855184;
   w2[167] := -0.2678719;
   w2[168] := 0.3169011;
   w2[169] := 0.0269058;
   w2[170] := 0.139307;
   w2[171] := 0.2074015;
   w2[172] := 0.044378;
   w2[173] := 0.3336064;
   w2[174] := -0.1919886;
   w2[175] := 0.0043234;
   w2[176] := 0.5604227;
   w2[177] := -0.1127777;
   w2[178] := -0.3165137;
   w2[179] := 0.2200206;
   w2[180] := -0.2163805;
   w2[181] := -0.239696;
   w2[182] := 0.1728129;
   w2[183] := -0.1887252;
   w2[184] := 0.2727011;
   w2[185] := 0.1560453;
   w2[186] := 0.457509;
   w2[187] := -0.2272316;
   w2[188] := 0.3077642;
   w2[189] := 0.06774;
   w2[190] := -0.050842;
   w2[191] := 0.0844207;
   w2[192] := 0.2612096;
   w2[193] := -0.0461612;
   w2[194] := 0.196588;
   w2[195] := 0.1832603;
   w2[196] := -0.1259902;
   w2[197] := 0.4958175;
   w2[198] := 0.3578667;
   w2[199] := -0.2289235;
   w2[200] := 0.0412198;
   w2[201] := -0.1472023;
   w2[202] := 0.5003238;
   w2[203] := 0.2104491;
   w2[204] := -0.3506398;
   w2[205] := -0.7278167;
   w2[206] := -0.1053378;
   w2[207] := -0.6664331;
   w2[208] := 0.3304765;
   w2[209] := 0.1904697;
   w2[210] := -0.5255481;
   w2[211] := 0.3779066;
   w2[212] := 0.575013;
   w2[213] := -0.4405918;
   w2[214] := 0.0437819;
   w2[215] := 0.0799071;
   w2[216] := -0.3873571;
   w2[217] := -0.1107465;
   w2[218] := -0.2144487;
   w2[219] := -0.452094;
   w2[220] := -0.0942226;
   w2[221] := -0.1042965;
   w2[222] := -0.0900685;
   w2[223] := -0.0358909;
   w2[224] := 0.5961101;
   w2[225] := -0.0502036;
   w2[226] := -0.205787;
   w2[227] := 0.1793782;
   w2[228] := 0.0139435;
   w2[229] := 0.140426;
   w2[230] := -0.1710399;
   w2[231] := -0.1097762;
   w2[232] := 0.6955358;
   w2[233] := -0.0941478;
   w2[234] := -0.6882815;
   w2[235] := -0.2339452;
   w2[236] := -0.5887371;
   w2[237] := 0.0302498;
   w2[238] := 0.2707806;
   w2[239] := -0.6653628;
   w2[240] := 0.3887634;
   w2[241] := 0.1627363;
   w2[242] := 0.0122889;
   w2[243] := -0.4034282;
   w2[244] := 0.3380547;
   w2[245] := -0.0177897;
   w2[246] := -0.1635698;
   w2[247] := -0.1298062;
   w2[248] := 0.2896215;
   w2[249] := 0.1131524;
   w2[250] := -0.2054364;
   w2[251] := 0.0131579;
   w2[252] := -0.890228;
   w2[253] := -0.6914336;
   w2[254] := -0.8277874;
   w2[255] := 0.254033;
   w2[256] := 0.179194;
   w2[257] := 0.0266804;
   w2[258] := -0.1867425;
   w2[259] := 0.1680747;
   w2[260] := -1.05107;
   w2[261] := -0.5665534;
   w2[262] := -0.1247267;
   w2[263] := -0.053494;
   w2[264] := 0.23726;
   w2[265] := -0.584154;
   w2[266] := -0.2938985;
   w2[267] := 0.1965791;
   w2[268] := 0.5103638;
   w2[269] := -0.0550255;
   w2[270] := -1.126066;
   w2[271] := 0.0735265;
   w2[272] := -0.2777269;
   w2[273] := 0.3135782;
   w2[274] := 0.1041824;
   w2[275] := -0.1324059;
   w2[276] := -0.3669493;
   w2[277] := -0.2885313;
   w2[278] := -0.367729;
   w2[279] := 0.1541151;
   w2[280] := 0.1346243;
   w2[281] := 0.6931639;
   w2[282] := 0.3574378;
   w2[283] := -0.1421183;
   w2[284] := 0.2825844;
   w2[285] := 0.0992049;
   w2[286] := 0.3324718;
   w2[287] := 0.168798;
   w2[288] := 0.1662632;
   w2[289] := -0.5125447;
   w2[290] := 0.1457812;
   w2[291] := -0.2258452;
   w2[292] := -0.2428768;
   w2[293] := 0.2717957;
   w2[294] := 0.0867224;
   w2[295] := -0.2496022;
   w2[296] := 0.1867056;
   w2[297] := -0.4031086;
   w2[298] := 0.4832774;
   w2[299] := 0.2478154;
   w2[300] := 0.0475016;
   w2[301] := -0.1532699;
   w2[302] := -0.6021184;
   w2[303] := -0.4835578;
   w2[304] := 0.348039;
   w2[305] := -0.0061014;
   w2[306] := 0.2888969;
   w2[307] := 0.0215752;
   w2[308] := 0.0208341;
   w2[309] := 0.5199659;
   w2[310] := 0.3490263;
   w2[311] := -0.0288161;
   w2[312] := -0.068543;
   w2[313] := -0.1182679;
   w2[314] := 0.3420109;
   w2[315] := -0.0353185;
   w2[316] := -0.1071727;
   w2[317] := -0.7671919;
   w2[318] := -0.3097001;
   w2[319] := 0.0119445;
   w2[320] := 0.1677119;
   w2[321] := -0.0187103;
   w2[322] := -0.0632623;
   w2[323] := 0.3558021;
   w2[324] := 0.4361037;
   w2[325] := -0.5477799;
   w2[326] := 0.1640894;
   w2[327] := 0.3476633;
   w2[328] := -0.2296589;
   w2[329] := -0.0005878;
   w2[330] := -0.1486427;
   w2[331] := -0.1145124;
   w2[332] := 0.1935411;
   w2[333] := -0.0498571;
   w2[334] := 0.007102;
   w2[335] := 0.1442345;
   w2[336] := -0.7647343;
   w2[337] := -0.7446802;
   w2[338] := -0.8727151;
   w2[339] := 0.3649753;
   w2[340] := 0.182284;
   w2[341] := 0.2168968;
   w2[342] := -0.3110866;
   w2[343] := 0.2285281;
   w2[344] := -0.8572159;
   w2[345] := -0.253249;
   w2[346] := -0.1099993;
   w2[347] := -0.1176312;
   w2[348] := 0.3110442;
   w2[349] := -0.0493409;
   w2[350] := 0.0371198;
   w2[351] := 0.2336326;
   w2[352] := 0.2238284;
   w2[353] := -0.0283122;
   w2[354] := -0.1704783;
   w2[355] := 0.0574998;
   w2[356] := -0.2733924;
   w2[357] := 0.0665076;
   w2[358] := 0.0320759;
   w2[359] := -0.1596949;
   w2[360] := -0.2385386;
   w2[361] := -0.2472534;
   w2[362] := -0.1323308;
   w2[363] := 0.1628101;
   w2[364] := 0.4503315;
   w2[365] := 0.1501646;
   w2[366] := 0.1143262;
   w2[367] := 0.023902;
   w2[368] := 0.0073025;
   w2[369] := 0.1456288;
   w2[370] := -0.3334046;
   w2[371] := 0.0482971;
   w2[372] := 0.4867398;
   w2[373] := -0.4917139;
   w2[374] := -0.6253324;
   w2[375] := -0.1267435;
   w2[376] := -0.2428251;
   w2[377] := -0.2196695;
   w2[378] := 0.1073758;
   w2[379] := 0.0506342;
   w2[380] := 0.4630886;
   w2[381] := -0.1982542;
   w2[382] := 0.3006389;
   w2[383] := -0.1852189;
   w2[384] := 0.1438557;
   w2[385] := 0.2112408;
   w2[386] := -0.1989525;
   w2[387] := -0.5165743;
   w2[388] := 0.2818699;
   w2[389] := 0.1988503;
   w2[390] := 0.0899179;
   w2[391] := 0.0992274;
   w2[392] := 0.3425773;
   w2[393] := -0.0475926;
   w2[394] := 0.0767343;
   w2[395] := 0.0394692;
   w2[396] := 0.1684201;
   w2[397] := -0.1340467;
   w2[398] := -0.3633062;
   w2[399] := -0.3210598;
   w2[400] := 0.5503753;
   w2[401] := 0.2680424;
   w2[402] := -0.2979992;
   w2[403] := -0.3373846;
   w2[404] := -0.2860682;
   w2[405] := 0.0260232;
   w2[406] := -0.1706583;
   w2[407] := -0.4802254;
   w2[408] := 0.1432097;
   w2[409] := 0.2762946;
   w2[410] := -0.3853753;
   w2[411] := -0.4026088;
   w2[412] := 0.3293981;
   w2[413] := 0.031134;
   w2[414] := 0.1150283;
   w2[415] := 0.032845;
   w2[416] := 0.1377832;
   w2[417] := 0.2112923;
   w2[418] := 0.0084318;
   w2[419] := 0.0693316;
   w2[420] := 0.0293756;
   w2[421] := 0.1045898;
   w2[422] := 0.2854653;
   w2[423] := 0.0997073;
   w2[424] := 0.1003512;
   w2[425] := -0.0351206;
   w2[426] := 0.4399726;
   w2[427] := 0.2780291;
   w2[428] := -0.0804132;
   w2[429] := 0.7397832;
   w2[430] := 0.7269561;
   w2[431] := 0.2094024;
   w2[432] := -0.2141474;
   w2[433] := 0.2012126;
   w2[434] := -0.2318728;
   w2[435] := -0.1762547;
   w2[436] := -0.0704646;
   w2[437] := 0.2301458;
   w2[438] := -0.0323121;
   w2[439] := 0.1872706;
   w2[440] := 0.4350786;
   w2[441] := 0.266441;
   w2[442] := 0.2541361;
   w2[443] := 0.1549129;
   w2[444] := -0.1279981;
   w2[445] := -0.1567508;
   w2[446] := 0.1148285;
   w2[447] := -0.2802774;
   g4[0] := -3.0;
   g4[1] := -2.571429;
   g4[2] := -2.142857;
   g4[3] := -1.714286;
   g4[4] := -1.285714;
   g4[5] := -0.8571429;
   g4[6] := -0.4285714;
   g4[8] := 0.4285714;
   g4[9] := 0.8571429;
   g4[10] := 1.285714;
   g4[11] := 1.714286;
   g4[12] := 2.142857;
   g4[13] := 2.571429;
   g4[14] := 3.0;
   t5[0] := 0.0969458;
   t5[1] := 0.0988391;
   t5[2] := 0.1005933;
   t5[3] := 0.1022003;
   t5[4] := 0.1036521;
   t5[5] := 0.1049404;
   t5[6] := 0.1060571;
   t5[7] := 0.1069942;
   t5[8] := 0.1077435;
   t5[9] := 0.1082969;
   t5[10] := 0.1086466;
   t5[11] := 0.1087928;
   t5[12] := 0.1087441;
   t5[13] := 0.1085093;
   t5[14] := 0.1080972;
   t5[15] := 0.0692292;
   t5[16] := 0.0677745;
   t5[17] := 0.0662769;
   t5[18] := 0.064728;
   t5[19] := 0.0631196;
   t5[20] := 0.0614434;
   t5[21] := 0.059691;
   t5[22] := 0.0578541;
   t5[23] := 0.0559245;
   t5[24] := 0.0538938;
   t5[25] := 0.051754;
   t5[26] := 0.0495057;
   t5[27] := 0.0471581;
   t5[28] := 0.0447209;
   t5[29] := 0.0422036;
   t5[30] := 0.0769506;
   t5[31] := 0.0739251;
   t5[32] := 0.0708925;
   t5[33] := 0.0678603;
   t5[34] := 0.0648361;
   t5[35] := 0.0618276;
   t5[36] := 0.0588422;
   t5[37] := 0.0558878;
   t5[38] := 0.0529718;
   t5[39] := 0.0501018;
   t5[40] := 0.0472854;
   t5[41] := 0.0445256;
   t5[42] := 0.0418212;
   t5[43] := 0.0391708;
   t5[44] := 0.036573;
   t5[45] := 0.0185666;
   t5[46] := 0.0167048;
   t5[47] := 0.0148043;
   t5[48] := 0.0128722;
   t5[49] := 0.0109158;
   t5[50] := 0.0089421;
   t5[51] := 0.0069585;
   t5[52] := 0.0049719;
   t5[53] := 0.0029896;
   t5[54] := 0.0010187;
   t5[55] := -0.0009336;
   t5[56] := -0.0028601;
   t5[57] := -0.0047537;
   t5[58] := -0.0066073;
   t5[59] := -0.0084138;
   t5[60] := -0.0480992;
   t5[61] := -0.0413032;
   t5[62] := -0.0343254;
   t5[63] := -0.0271627;
   t5[64] := -0.0198121;
   t5[65] := -0.0122706;
   t5[66] := -0.0045353;
   t5[67] := 0.003397;
   t5[68] := 0.0115292;
   t5[69] := 0.0198644;
   t5[70] := 0.028405;
   t5[71] := 0.0371425;
   t5[72] := 0.0460565;
   t5[73] := 0.0551263;
   t5[74] := 0.0643312;
   t5[75] := 0.0416106;
   t5[76] := 0.0386293;
   t5[77] := 0.0355967;
   t5[78] := 0.032509;
   t5[79] := 0.0293625;
   t5[80] := 0.0261533;
   t5[81] := 0.0228775;
   t5[82] := 0.0195314;
   t5[83] := 0.0161111;
   t5[84] := 0.0126127;
   t5[85] := 0.0090329;
   t5[86] := 0.005375;
   t5[87] := 0.0016502;
   t5[88] := -0.0021304;
   t5[89] := -0.0059555;
   t5[90] := 0.040686;
   t5[91] := 0.031406;
   t5[92] := 0.0221584;
   t5[93] := 0.0129649;
   t5[94] := 0.0038467;
   t5[95] := -0.0051745;
   t5[96] := -0.0140773;
   t5[97] := -0.0228401;
   t5[98] := -0.0314415;
   t5[99] := -0.03986;
   t5[100] := -0.0480745;
   t5[101] := -0.0560725;
   t5[102] := -0.0638503;
   t5[103] := -0.0714046;
   t5[104] := -0.0787324;
   t5[105] := 0.0090538;
   t5[106] := 0.0118105;
   t5[107] := 0.0144813;
   t5[108] := 0.0170639;
   t5[109] := 0.019556;
   t5[110] := 0.0219552;
   t5[111] := 0.0242594;
   t5[112] := 0.0264662;
   t5[113] := 0.0285733;
   t5[114] := 0.0305785;
   t5[115] := 0.0324795;
   t5[116] := 0.0342752;
   t5[117] := 0.0359658;
   t5[118] := 0.0375512;
   t5[119] := 0.0390318;
   t5[120] := 0.0821998;
   t5[121] := 0.0801324;
   t5[122] := 0.0780161;
   t5[123] := 0.0758536;
   t5[124] := 0.0736473;
   t5[125] := 0.0713999;
   t5[126] := 0.0691138;
   t5[127] := 0.0667916;
   t5[128] := 0.0644359;
   t5[129] := 0.0620491;
   t5[130] := 0.0596339;
   t5[131] := 0.0571941;
   t5[132] := 0.0547352;
   t5[133] := 0.0522623;
   t5[134] := 0.049781;
   t5[135] := -0.0523619;
   t5[136] := -0.0494093;
   t5[137] := -0.0463022;
   t5[138] := -0.0430293;
   t5[139] := -0.0395791;
   t5[140] := -0.0359404;
   t5[141] := -0.0321018;
   t5[142] := -0.0280519;
   t5[143] := -0.0237793;
   t5[144] := -0.0192728;
   t5[145] := -0.0145215;
   t5[146] := -0.0095269;
   t5[147] := -0.004303;
   t5[148] := 0.0011352;
   t5[149] := 0.0067732;
   t5[150] := 0.0102707;
   t5[151] := 0.0063571;
   t5[152] := 0.0025329;
   t5[153] := -0.0011961;
   t5[154] := -0.0048241;
   t5[155] := -0.0083454;
   t5[156] := -0.0117542;
   t5[157] := -0.0150446;
   t5[158] := -0.018211;
   t5[159] := -0.0212476;
   t5[160] := -0.0241488;
   t5[161] := -0.0269126;
   t5[162] := -0.029541;
   t5[163] := -0.0320361;
   t5[164] := -0.0344;
   t5[165] := 0.0980121;
   t5[166] := 0.0995716;
   t5[167] := 0.1009058;
   t5[168] := 0.1020029;
   t5[169] := 0.1028509;
   t5[170] := 0.1034377;
   t5[171] := 0.1037513;
   t5[172] := 0.1037798;
   t5[173] := 0.1035112;
   t5[174] := 0.1029334;
   t5[175] := 0.102035;
   t5[176] := 0.100816;
   t5[177] := 0.0992884;
   t5[178] := 0.0974645;
   t5[179] := 0.095357;
   t5[180] := -0.0973992;
   t5[181] := -0.0943194;
   t5[182] := -0.0910766;
   t5[183] := -0.0876704;
   t5[184] := -0.0841003;
   t5[185] := -0.080366;
   t5[186] := -0.076467;
   t5[187] := -0.0724028;
   t5[188] := -0.068173;
   t5[189] := -0.0637771;
   t5[190] := -0.059215;
   t5[191] := -0.054491;
   t5[192] := -0.0496145;
   t5[193] := -0.0445951;
   t5[194] := -0.0394423;
   t5[195] := 0.0479108;
   t5[196] := 0.0463938;
   t5[197] := 0.0450368;
   t5[198] := 0.0438498;
   t5[199] := 0.0428428;
   t5[200] := 0.0420256;
   t5[201] := 0.0414083;
   t5[202] := 0.0410008;
   t5[203] := 0.0408131;
   t5[204] := 0.0408551;
   t5[205] := 0.0411363;
   t5[206] := 0.0416536;
   t5[207] := 0.0423913;
   t5[208] := 0.0433331;
   t5[209] := 0.0444624;
   t5[210] := 0.1111941;
   t5[211] := 0.1078871;
   t5[212] := 0.1045146;
   t5[213] := 0.1010781;
   t5[214] := 0.0975793;
   t5[215] := 0.0940199;
   t5[216] := 0.0904016;
   t5[217] := 0.086726;
   t5[218] := 0.0829947;
   t5[219] := 0.0792094;
   t5[220] := 0.0753718;
   t5[221] := 0.0714837;
   t5[222] := 0.0675472;
   t5[223] := 0.0635644;
   t5[224] := 0.0595373;
   t5[225] := -0.0148444;
   t5[226] := -0.0188319;
   t5[227] := -0.0227787;
   t5[228] := -0.0266817;
   t5[229] := -0.0305375;
   t5[230] := -0.0343429;
   t5[231] := -0.0380947;
   t5[232] := -0.0417897;
   t5[233] := -0.0454244;
   t5[234] := -0.0489958;
   t5[235] := -0.0525006;
   t5[236] := -0.0559371;
   t5[237] := -0.0593051;
   t5[238] := -0.0626045;
   t5[239] := -0.0658352;
   t5[240] := 0.1048705;
   t5[241] := 0.1052619;
   t5[242] := 0.1056781;
   t5[243] := 0.1061181;
   t5[244] := 0.1065808;
   t5[245] := 0.1070651;
   t5[246] := 0.1075699;
   t5[247] := 0.1080941;
   t5[248] := 0.1086367;
   t5[249] := 0.1091965;
   t5[250] := 0.1097724;
   t5[251] := 0.1103615;
   t5[252] := 0.1109593;
   t5[253] := 0.111561;
   t5[254] := 0.112162;
   t5[255] := 0.110168;
   t5[256] := 0.1074914;
   t5[257] := 0.1045742;
   t5[258] := 0.1014118;
   t5[259] := 0.0979995;
   t5[260] := 0.0943326;
   t5[261] := 0.0904064;
   t5[262] := 0.0862162;
   t5[263] := 0.0817574;
   t5[264] := 0.0770252;
   t5[265] := 0.0720154;
   t5[266] := 0.0667328;
   t5[267] := 0.0611919;
   t5[268] := 0.0554075;
   t5[269] := 0.0493943;
   t5[270] := 0.0740068;
   t5[271] := 0.0726272;
   t5[272] := 0.0712559;
   t5[273] := 0.0698956;
   t5[274] := 0.0685491;
   t5[275] := 0.0672189;
   t5[276] := 0.0659077;
   t5[277] := 0.0646183;
   t5[278] := 0.0633531;
   t5[279] := 0.0621149;
   t5[280] := 0.0609064;
   t5[281] := 0.0597273;
   t5[282] := 0.058575;
   t5[283] := 0.0574468;
   t5[284] := 0.0563398;
   t5[285] := 0.0339974;
   t5[286] := 0.0288029;
   t5[287] := 0.023595;
   t5[288] := 0.0183771;
   t5[289] := 0.0131526;
   t5[290] := 0.0079248;
   t5[291] := 0.0026971;
   t5[292] := -0.0025272;
   t5[293] := -0.0077446;
   t5[294] := -0.0129518;
   t5[295] := -0.0181454;
   t5[296] := -0.0233209;
   t5[297] := -0.0284728;
   t5[298] := -0.0335955;
   t5[299] := -0.0386833;
   t5[300] := 0.0620911;
   t5[301] := 0.0607191;
   t5[302] := 0.0590387;
   t5[303] := 0.0570417;
   t5[304] := 0.0547198;
   t5[305] := 0.0520647;
   t5[306] := 0.0490683;
   t5[307] := 0.0457222;
   t5[308] := 0.0420181;
   t5[309] := 0.0379479;
   t5[310] := 0.0335039;
   t5[311] := 0.0286934;
   t5[312] := 0.0235394;
   t5[313] := 0.0180654;
   t5[314] := 0.0122949;
   t5[315] := 0.1065427;
   t5[316] := 0.1071066;
   t5[317] := 0.1075431;
   t5[318] := 0.107845;
   t5[319] := 0.1080055;
   t5[320] := 0.1080177;
   t5[321] := 0.1078745;
   t5[322] := 0.107569;
   t5[323] := 0.1070943;
   t5[324] := 0.1064434;
   t5[325] := 0.1056096;
   t5[326] := 0.1045918;
   t5[327] := 0.1033945;
   t5[328] := 0.1020227;
   t5[329] := 0.1004812;
   t5[330] := -0.0022573;
   t5[331] := 0.0009967;
   t5[332] := 0.0041721;
   t5[333] := 0.0072579;
   t5[334] := 0.0102434;
   t5[335] := 0.0131175;
   t5[336] := 0.0158695;
   t5[337] := 0.0184885;
   t5[338] := 0.0209636;
   t5[339] := 0.0232839;
   t5[340] := 0.025439;
   t5[341] := 0.0274273;
   t5[342] := 0.0292566;
   t5[343] := 0.030935;
   t5[344] := 0.0324708;
   t5[345] := 0.0238222;
   t5[346] := 0.0248892;
   t5[347] := 0.0260044;
   t5[348] := 0.0271786;
   t5[349] := 0.0284228;
   t5[350] := 0.0297477;
   t5[351] := 0.031164;
   t5[352] := 0.0326828;
   t5[353] := 0.0343147;
   t5[354] := 0.0360705;
   t5[355] := 0.0379608;
   t5[356] := 0.0399854;
   t5[357] := 0.0421339;
   t5[358] := 0.0443951;
   t5[359] := 0.046758;
   t5[360] := 0.0368159;
   t5[361] := 0.0420822;
   t5[362] := 0.0473928;
   t5[363] := 0.0527457;
   t5[364] := 0.0581387;
   t5[365] := 0.0635699;
   t5[366] := 0.069037;
   t5[367] := 0.074538;
   t5[368] := 0.0800708;
   t5[369] := 0.0856332;
   t5[370] := 0.0912231;
   t5[371] := 0.096835;
   t5[372] := 0.1024601;
   t5[373] := 0.1080894;
   t5[374] := 0.1137142;
   t5[375] := 0.006496;
   t5[376] := 0.003554;
   t5[377] := 0.0006008;
   t5[378] := -0.0023534;
   t5[379] := -0.0052987;
   t5[380] := -0.0082251;
   t5[381] := -0.0111224;
   t5[382] := -0.0139808;
   t5[383] := -0.0167902;
   t5[384] := -0.0195405;
   t5[385] := -0.0222221;
   t5[386] := -0.0248314;
   t5[387] := -0.0273713;
   t5[388] := -0.0298452;
   t5[389] := -0.0322563;
   t5[390] := 0.1115208;
   t5[391] := 0.1148185;
   t5[392] := 0.1180112;
   t5[393] := 0.1210973;
   t5[394] := 0.1240754;
   t5[395] := 0.1269439;
   t5[396] := 0.1297014;
   t5[397] := 0.1323464;
   t5[398] := 0.1348774;
   t5[399] := 0.1372929;
   t5[400] := 0.1395914;
   t5[401] := 0.1417692;
   t5[402] := 0.1438208;
   t5[403] := 0.1457406;
   t5[404] := 0.1475227;
   t5[405] := 0.0927025;
   t5[406] := 0.0939897;
   t5[407] := 0.0951551;
   t5[408] := 0.0961991;
   t5[409] := 0.0971219;
   t5[410] := 0.097924;
   t5[411] := 0.0986054;
   t5[412] := 0.0991667;
   t5[413] := 0.0996081;
   t5[414] := 0.0999298;
   t5[415] := 0.1001323;
   t5[416] := 0.100218;
   t5[417] := 0.1001915;
   t5[418] := 0.1000572;
   t5[419] := 0.0998198;
   t5[420] := 0.1446864;
   t5[421] := 0.1460695;
   t5[422] := 0.1473257;
   t5[423] := 0.1484532;
   t5[424] := 0.1494499;
   t5[425] := 0.1503137;
   t5[426] := 0.1510427;
   t5[427] := 0.1516349;
   t5[428] := 0.1520882;
   t5[429] := 0.1524006;
   t5[430] := 0.1525704;
   t5[431] := 0.1525994;
   t5[432] := 0.1524938;
   t5[433] := 0.1522598;
   t5[434] := 0.1519035;
   t5[435] := -0.0403738;
   t5[436] := -0.0373444;
   t5[437] := -0.0341651;
   t5[438] := -0.0308276;
   t5[439] := -0.0273232;
   t5[440] := -0.0236437;
   t5[441] := -0.0197805;
   t5[442] := -0.0157252;
   t5[443] := -0.0114694;
   t5[444] := -0.0070046;
   t5[445] := -0.0023229;
   t5[446] := 0.0025711;
   t5[447] := 0.0076596;
   t5[448] := 0.0129246;
   t5[449] := 0.018348;
   t5[450] := 0.1207302;
   t5[451] := 0.1224805;
   t5[452] := 0.1241813;
   t5[453] := 0.1258319;
   t5[454] := 0.1274316;
   t5[455] := 0.1289798;
   t5[456] := 0.1304759;
   t5[457] := 0.131919;
   t5[458] := 0.1333087;
   t5[459] := 0.1346441;
   t5[460] := 0.1359247;
   t5[461] := 0.1371484;
   t5[462] := 0.138312;
   t5[463] := 0.1394122;
   t5[464] := 0.1404457;
   t5[465] := 0.2641891;
   t5[466] := 0.2561393;
   t5[467] := 0.2478748;
   t5[468] := 0.2394127;
   t5[469] := 0.2307699;
   t5[470] := 0.2219633;
   t5[471] := 0.2130101;
   t5[472] := 0.2039271;
   t5[473] := 0.1947314;
   t5[474] := 0.1854398;
   t5[475] := 0.1760694;
   t5[476] := 0.1666338;
   t5[477] := 0.1571439;
   t5[478] := 0.1476101;
   t5[479] := 0.138043;
